(* IEC 61131-3 sources: SmartHomeNew/, 564 files *)

(* ---- E_Heating_Policy_Mode.typ ---- *)
TYPE E_Heating_Policy_Mode :
(
    HPM_NORMAL,
    HPM_DEGRADED,
    HPM_FREEZE_PROTECT,
    HPM_MAINTENANCE,
    HPM_SAFETY_BLOCK,
    HPM_FAULT_ISOLATION
);
END_TYPE

(* ---- E_Modbus_SysCom_Backend_State.dut ---- *)
TYPE E_Modbus_SysCom_Backend_State :
(
    MB_SYSCOM_CLOSED := 0,
    MB_SYSCOM_OPENING := 1,
    MB_SYSCOM_ONLINE := 2,
    MB_SYSCOM_ERROR := 3,
    MB_SYSCOM_RECONNECT_WAIT := 4
);
END_TYPE

(* ---- E_Recovery_Phase.dut ---- *)
{attribute 'strict'}
TYPE E_Recovery_Phase :
(
    IDLE := 0,
    STABILIZING := 1,
    WAIT_MANUAL_CONFIRM := 2,
    RECOVERING := 3,
    COOLDOWN := 4,
    ABORTED := 5
) USINT;
END_TYPE

(* ---- E_Runtime_Observer_Deny_Reason.typ ---- *)
TYPE E_Runtime_Observer_Deny_Reason :
(
    RODR_NONE := 0,
    RODR_NO_ENABLE_REQUEST := 10,
    RODR_BOOTSTRAP_DISABLED := 100,
    RODR_PASSIVE_MODE_DISABLED := 110,
    RODR_READONLY_MODE_DISABLED := 120,
    RODR_GOVERNANCE_UNLOCKED := 130,
    RODR_RUNTIME_AUTHORITY_ENABLED := 140,
    RODR_WRITABLE_EXPORTS_ENABLED := 150
);
END_TYPE

(* ---- E_Safety_Mode.dut ---- *)
{attribute 'strict'}
TYPE E_Safety_Mode :
(
    NORMAL := 0,
    FIRE := 1,
    GAS := 2,
    WATER_LEAK := 3,
    GLOBAL_STOP := 4
) USINT;
END_TYPE

(* ---- E_SCENARIO_TYPE.dut ---- *)
{attribute 'strict'}
TYPE E_SCENARIO_TYPE :
(
    SCENARIO_NONE := 0,
    SCENARIO_MORNING := 1,
    SCENARIO_EVENING := 2,
    SCENARIO_AWAY := 3,
    SCENARIO_PARTY := 4,
    SCENARIO_SLEEP := 5,
    SCENARIO_EMERGENCY := 6,
    SCENARIO_PRESENCE := 7
) USINT;
END_TYPE

(* ---- E_System_Reason_Code.dut ---- *)
{attribute 'strict'}
TYPE E_System_Reason_Code :
(
    REASON_NONE := 0,
    REASON_USER := 1,
    REASON_SAFETY := 2,
    REASON_AUTOMATION := 3,
    REASON_INTERNAL := 4,
    REASON_SCENARIO_VENT_BOOST := 5
) USINT;
END_TYPE

(* ---- E_Trace_Layer.dut ---- *)
{attribute 'strict'}
TYPE E_Trace_Layer :
(
    TRACE_SYSTEM := 0,
    TRACE_SAFETY := 1,
    TRACE_HEATING := 2,
    TRACE_IO := 3,
    TRACE_SCENARIO := 4,
    TRACE_USER := 5
) USINT;
END_TYPE

(* ---- E_Trace_Source.dut ---- *)
{attribute 'strict'}
TYPE E_Trace_Source :
(
    SRC_MAIN := 0,
    SRC_IO := 1,
    SRC_DIAGNOSTICS := 2,
    SRC_HEATING := 3,
    SRC_SCENARIO := 4
) USINT;
END_TYPE

(* ---- E_Valve_Test_Result.dut ---- *)
{attribute 'strict'}
TYPE E_Valve_Test_Result :
(
    TEST_RESULT_NONE := 0,
    TEST_RESULT_PASSED := 1,
    TEST_RESULT_CURRENT_DEVIATION := 2,
    TEST_RESULT_TIME_DEVIATION := 3,
    TEST_RESULT_STALL := 4,
    TEST_RESULT_LIMIT_SWITCH_FAIL := 5,
    TEST_RESULT_ABORTED := 6
) USINT;
END_TYPE

(* ---- GVL_EXPLAINABILITY.gvl ---- *)
TYPE E_System_Reason_Code :
(
    REASON_NONE,
    REASON_FIRE,
    REASON_GAS,
    REASON_WATER_LEAK,
    REASON_GLOBAL_STOP,
    REASON_EVACUATION,
    REASON_RECOVERY_ACTIVE,
    REASON_SAFETY,
    REASON_USER_REQUEST,
    REASON_COMMAND_CLAMP,
    REASON_DOMAIN_PROJECTION,
    REASON_SCENARIO_NIGHT,
    REASON_SCENARIO_COMFORT,
    REASON_SCENARIO_ENERGY_SAVE,
    REASON_SCENARIO_AWAY,
    REASON_SCENARIO_PREHEAT,
    REASON_SCENARIO_ACCESS_SECURE,
    REASON_SCENARIO_VENT_BOOST
);
END_TYPE

VAR_GLOBAL
    G_Last_Global_Reason_Code : E_System_Reason_Code := REASON_NONE;
    G_Last_Global_Reason_Text : STRING(255) := 'No active reason';
    G_Last_Safety_Mode : E_Safety_Mode := NORMAL;
    G_Last_Recovery_Phase : E_Recovery_Phase := IDLE;
    G_Last_Command_Source : STRING(80) := '';
    G_Last_Domain_Affected : STRING(80) := '';
    G_Last_Output_Affected : STRING(80) := '';
    G_Last_Update_MS : UDINT := 0;

    G_Behavior_Why_Active : STRING(255) := '';
    G_Heating_Why_Blocked : STRING(255) := '';
    G_Vent_Why_Stopped : STRING(255) := '';
    G_Water_Why_Closed : STRING(255) := '';
    G_Access_Why_Opened : STRING(255) := '';

    // Decision chain for HMI / engineering debug.
    G_Reason_Chain_Safety : STRING(80) := 'NORMAL';
    G_Reason_Chain_Behavior : STRING(120) := 'No behavior scenario active';
    G_Reason_Chain_Command : STRING(120) := 'Command OK';
    G_Reason_Chain_Output : STRING(120) := 'Outputs projected';
    G_Reason_Chain_Full : STRING(255) := 'NORMAL -> No behavior scenario active -> Command OK -> Outputs projected';
END_VAR

(* ---- GVL_SAFETY_RECOVERY.gvl ---- *)
TYPE E_Recovery_Phase :
(
    IDLE,
    STABILIZING,
    WAIT_MANUAL_CONFIRM,
    RECOVERING,
    COOLDOWN,
    ABORTED
);
END_TYPE

VAR_GLOBAL
    G_Recovery_Phase : E_Recovery_Phase := IDLE;
    G_Recovery_Active : BOOL := FALSE;
    G_Recovery_Requested : BOOL := FALSE;
    G_Recovery_Manual_Confirm : BOOL := FALSE;
    G_Recovery_Start_MS : UDINT := 0;
    G_Recovery_Stable_Since_MS : UDINT := 0;
    G_Recovery_Cooldown_Start_MS : UDINT := 0;
    G_Recovery_Exit_Allowed : BOOL := FALSE;
    G_Recovery_Abort_Reason : INT := 0; // 0=none, 1=safety active, 2=confidence low, 3=timeout
END_VAR

(* ---- GVL_SEMANTIC_EXECUTION_CONTROL.gvl ---- *)
TYPE E_SEMANTIC_EXECUTION_PATH : (
    FAST_PATH,
    NORMAL_PATH,
    DEFERRED_PATH,
    BACKGROUND_PATH
);
END_TYPE

VAR_GLOBAL
    // Semantic execution governance.
    Semantic_Execution_Control_Active : BOOL := TRUE;
    Semantic_Execution_Control_ReadOnly : BOOL := TRUE;

    // Canonical verification domains.
    Temporal_Verification_Domain_Active : BOOL := TRUE;
    Authority_Verification_Domain_Active : BOOL := TRUE;
    Physical_Verification_Domain_Active : BOOL := TRUE;
    Runtime_Verification_Domain_Active : BOOL := TRUE;
    Survivability_Verification_Domain_Active : BOOL := TRUE;

    // Deterministic semantic scheduling.
    Safety_Execution_Path : E_SEMANTIC_EXECUTION_PATH := FAST_PATH;
    Physical_Verification_Path : E_SEMANTIC_EXECUTION_PATH := FAST_PATH;
    Runtime_Verification_Path : E_SEMANTIC_EXECUTION_PATH := NORMAL_PATH;
    Diagnostics_Execution_Path : E_SEMANTIC_EXECUTION_PATH := DEFERRED_PATH;
    Trend_Analytics_Execution_Path : E_SEMANTIC_EXECUTION_PATH := BACKGROUND_PATH;

    // Semantic execution collapse prevention.
    Semantic_Execution_Fragmentation_Risk : BOOL := FALSE;
    Semantic_Cascade_Amplification_Risk : BOOL := FALSE;
    Semantic_Complexity_Ceiling_Reached : BOOL := FALSE;

    // Runtime semantic limits.
    Semantic_Chain_Depth_Limit_Reached : BOOL := FALSE;
    Verification_Fanout_Limit_Reached : BOOL := FALSE;
    Observability_Fanout_Limit_Reached : BOOL := FALSE;
    Lifecycle_Transition_Limit_Reached : BOOL := FALSE;

    // Runtime-governed complexity ceiling.
    Autonomous_Complexity_Ceiling_Enforced : BOOL := FALSE;
    Semantic_Scheduler_Active : BOOL := TRUE;

    Semantic_Execution_Control_Epoch : UDINT := 0;
END_VAR

(* ---- GVL_TRACE.gvl ---- *)
TYPE E_Trace_Layer :
(
    TRACE_SENSOR,
    TRACE_SCENARIO,
    TRACE_INTENT,
    TRACE_COMMAND,
    TRACE_DOMAIN,
    TRACE_IO,
    TRACE_SAFETY,
    TRACE_RECOVERY
);
END_TYPE

TYPE E_Trace_Source :
(
    SRC_NONE,
    SRC_SENSOR,
    SRC_USER,
    SRC_SCENARIO,
    SRC_SAFETY,
    SRC_RECOVERY,
    SRC_COMMAND,
    SRC_DOMAIN,
    SRC_IO
);
END_TYPE

TYPE ST_Trace_Entry :
STRUCT
    Timestamp_MS : UDINT;
    Layer : E_Trace_Layer;
    Source : E_Trace_Source;
    Reason_Code : E_System_Reason_Code;
    Value_Bool : BOOL;
    Value_Real : REAL;
    Text : STRING(120);
END_STRUCT
END_TYPE

VAR_GLOBAL
    G_Trace_Buffer : ARRAY[1..200] OF ST_Trace_Entry;
    G_Trace_Write_Index : INT := 1;
    G_Trace_Enabled : BOOL := TRUE;
END_VAR

(* ---- ST_Astro_Time.dut ---- *)
{attribute 'pack_mode' := '1'}
TYPE ST_Astro_Time :
STRUCT
    sunrise_ms : UDINT := 0;
    sunset_ms : UDINT := 0;
    is_daylight : BOOL := FALSE;
END_STRUCT
END_TYPE

(* ---- ST_BlackBox_Record.dut ---- *)
{attribute 'pack_mode' := '1'}
TYPE ST_BlackBox_Record :
STRUCT
    Timestamp : UDINT;
    Gas_Methane_LEL : REAL;
    Gas_CO_PPM : REAL;
    Flood_Active : BOOL;
    Fire_Active : BOOL;
    Valve_Gas_Status : BYTE;
    Valve_Water_Status : BYTE;
    PLC_Active_ID : BYTE;
    System_Mode : BYTE; // Encoded E_System_Operating_Mode for diagnostics
    First_Fault_Type : BYTE; // 1=IO,2=Sensor,3=Comm,4=Subsystem
    First_Fault_Source : BYTE; // 1=Heating,2=DHW,3=Ventilation,4=Lighting,5=Access
    First_Fault_Active : BOOL;
    System_Severity : BYTE;
    Root_Cause      : BYTE;
    Watchdog_Fault  : BOOL; // Latched root cause active

END_STRUCT
END_TYPE

(* ---- ST_Boiler_Status.dut ---- *)
{attribute 'pack_mode' := '1'}
TYPE ST_Boiler_Status :
STRUCT
    Active : BOOL;
    Running : BOOL;
    Warning : BOOL;
    Error : BOOL;
    Error_ID : WORD;

    // Boiler thermal/runtime information
    Power_Percent : REAL;
    Current_Power : REAL;
    Work_Seconds : UDINT;
    Work_Hours : REAL;
    Resource_Percent : REAL := 100.0;
    Last_Start : DT;

    // OpenTherm transport observability
    OT_Online : BOOL;
    OT_Command_Valid : BOOL;
    OT_Transport_Degraded : BOOL;
    OT_Adapter_Error : BOOL;

    // Semantic cascade/explainability state
    Available : BOOL;
    Selected_By_Cascade : BOOL;
    Flame_Missing : BOOL;
    Transport_Missing : BOOL;
    Ignition_Timeout : BOOL;
    Degraded : BOOL;
END_STRUCT
END_TYPE

(* ---- ST_Config_Activation_State.dut ---- *)
TYPE ST_Config_Activation_State :
STRUCT
    Runtime_Valid : BOOL;
    Runtime_System_Time_MS : UDINT;

    Active_Version : UDINT;
    Staged_Version : UDINT;
    Previous_Stable_Version : UDINT;

    Staged_Config_Valid : BOOL;
    Activation_Requested : BOOL;
    Activation_Allowed : BOOL;
    Activation_Blocked : BOOL;
    Rollback_Requested : BOOL;
    Rollback_Available : BOOL;
    Rollback_Active : BOOL;

    Config_Quarantine_Active : BOOL;
    Migration_Required : BOOL;
    Migration_Compatible : BOOL;

    Status_Code : UINT;
    Status_Text : STRING(160);
END_STRUCT
END_TYPE

(* ---- ST_Debug_Log_Record.dut ---- *)
{attribute 'pack_mode' := '1'}
TYPE ST_Debug_Log_Record :
STRUCT
    timestamp_ms : UDINT;
    level : BYTE; // E_Debug_Log_Level
    source_id : BYTE;
    event_code : WORD;
    value_int : UDINT;
    value_real : REAL;
    text : STRING(80);
    crc32 : DWORD;
END_STRUCT
END_TYPE

(* ---- ST_Distributed_Projection_Ownership.dut ---- *)
TYPE ST_Distributed_Projection_Ownership :
STRUCT
    Ownership_Valid : BOOL;
    Runtime_System_Time_MS : UDINT;

    Projection_Id : UINT;
    Projection_Class : UINT;

    Owner_Controller_Id : UINT;
    Owner_Runtime_Node_Id : UINT;
    Owner_Authority_Domain_Id : UINT;

    Ownership_Granted : BOOL;
    Ownership_Revoked : BOOL;
    Ownership_Conflict : BOOL;
    Ownership_Stale : BOOL;

    Projection_Active : BOOL;
    Projection_Blocked : BOOL;

    Distributed_Execution_Allowed : BOOL;
    Distributed_Recovery_Allowed : BOOL;

    Status_Code : UINT;
    Status_Text : STRING(160);
END_STRUCT
END_TYPE

(* ---- ST_Distributed_Runtime_Node_State.dut ---- *)
TYPE ST_Distributed_Runtime_Node_State :
STRUCT
    Runtime_Valid : BOOL;
    Runtime_System_Time_MS : UDINT;

    Controller_Id : UINT;
    Runtime_Node_Id : UINT;
    Authority_Domain_Id : UINT;
    Topology_Domain_Id : UINT;

    Node_Online : BOOL;
    Node_Degraded : BOOL;
    Node_Quarantined : BOOL;
    Node_Backup_Mode : BOOL;
    Node_Observer_Mode : BOOL;

    Authority_Allowed : BOOL;
    Authority_Revoked : BOOL;
    Authority_Master : BOOL;
    Authority_Backup : BOOL;

    Replication_Healthy : BOOL;
    Replication_Timeout : BOOL;
    Split_Brain_Suspected : BOOL;

    Restart_Continuity_Valid : BOOL;
    Quarantine_State_Replicated : BOOL;
    Recovery_State_Replicated : BOOL;

    Status_Code : UINT;
    Status_Text : STRING(160);
END_STRUCT
END_TYPE

(* ---- ST_Distributed_Topology_Domain.dut ---- *)
TYPE ST_Distributed_Topology_Domain :
STRUCT
    Domain_Valid : BOOL;
    Domain_Id : UINT;
    Controller_Id : UINT;
    Runtime_Node_Id : UINT;

    Authority_Owner : BOOL;
    Backup_Owner : BOOL;
    Observer_Only : BOOL;

    Domain_Online : BOOL;
    Domain_Degraded : BOOL;
    Domain_Quarantined : BOOL;

    Cross_Node_Dependencies : BOOL;
    Remote_Valve_Group_Required : BOOL;
    Remote_Recovery_Required : BOOL;

    Distributed_Path_Valid : BOOL;
    Distributed_Projection_Allowed : BOOL;

    Status_Code : UINT;
    Status_Text : STRING(160);
END_STRUCT
END_TYPE

(* ---- ST_EVENT.dut ---- *)
TYPE ST_EVENT :
STRUCT
    Event_ID    : UDINT;
    Event_Type  : UINT;
    Timestamp   : UDINT;
    Param1      : UDINT;
    Param2      : UDINT;
END_STRUCT
END_TYPE

(* ---- ST_Flood_Config.dut ---- *)
{attribute 'pack_mode' := '1'}
TYPE ST_Flood_Config :
STRUCT
    Emergency_Two_Stage_Enabled : BOOL := TRUE;
    Valve_Test_Period_Days : UINT := 7;
    Current_Threshold_MA : REAL := 500.0;
    sensor_to_valve_map : ARRAY[1..GVL_CONSTANTS.C_MAX_FLOOD_SENSORS] OF INT := [1, 1, 1, 1, 2, 2, 2, 2, 3, 3, 3, 3]; // 1: ХВС, 2: ГВС, 3: Оба
END_STRUCT
END_TYPE

(* ---- ST_Heating_Command.st ---- *)
TYPE ST_Heating_Command :
STRUCT
    Enable              : BOOL;
    Target_Temperature  : REAL;
    Priority            : INT; // higher = stronger
END_STRUCT
END_TYPE

(* ---- ST_Heating_Runtime_Adaptive_Intelligence.dut ---- *)
TYPE ST_Heating_Runtime_Adaptive_Intelligence :
STRUCT
    // ======================================================
    // Adaptive lifecycle
    // ======================================================
    Intelligence_Active : BOOL;
    Intelligence_Degraded : BOOL;
    Intelligence_Critical : BOOL;

    // ======================================================
    // Adaptive supervision confidence
    // ======================================================
    Supervision_Confidence : UINT;
    Confidence_Degraded : BOOL;

    // ======================================================
    // Adaptive runtime risk
    // ======================================================
    Adaptive_Runtime_Risk : UINT;
    Adaptive_Runtime_Stability : UINT;

    // ======================================================
    // Adaptive anomaly weighting
    // ======================================================
    Runtime_Anomaly_Weight : UINT;
    Cascade_Anomaly_Weight : UINT;
    OpenTherm_Anomaly_Weight : UINT;
    Diagnostics_Anomaly_Weight : UINT;

    // ======================================================
    // Predictive correlation weighting
    // ======================================================
    Predictive_Correlation_Score : UINT;
    Predictive_Correlation_Degraded : BOOL;

    // ======================================================
    // Adaptive integrity
    // ======================================================
    Sequencing_Confidence : UINT;
    Ownership_Confidence : UINT;
    Synchronization_Confidence : UINT;

    // ======================================================
    // Adaptive status
    // ======================================================
    Status_Code : UINT;
    Status_Text : STRING(128);
END_STRUCT
END_TYPE

(* ---- ST_Heating_Runtime_Blackbox_Timeline.dut ---- *)
TYPE ST_Heating_Runtime_Blackbox_Timeline :
STRUCT
    // ======================================================
    // Blackbox events
    // ======================================================
    Events : ARRAY[1..256] OF ST_Heating_Runtime_Blackbox_Event;

    // ======================================================
    // Timeline state
    // ======================================================
    Write_Index : UINT;
    Event_Count : UINT;
    Timeline_Overflow : BOOL;

    // ======================================================
    // Runtime forensic state
    // ======================================================
    Reconstruction_Active : BOOL;
    Replay_Active : BOOL;
    Root_Cause_Reconstructed : BOOL;

    // ======================================================
    // Timeline integrity
    // ======================================================
    Sequencing_Valid : BOOL;
    Ownership_Valid : BOOL;
    Synchronization_Valid : BOOL;

    // ======================================================
    // Timeline status
    // ======================================================
    Status_Code : UINT;
    Status_Text : STRING(128);
END_STRUCT
END_TYPE

(* ---- ST_Heating_Runtime_Causality_Edge.dut ---- *)
TYPE ST_Heating_Runtime_Causality_Edge :
STRUCT
    // ======================================================
    // Edge topology
    // ======================================================
    Source_Node_ID : UINT;
    Target_Node_ID : UINT;

    // ======================================================
    // Edge lifecycle
    // ======================================================
    Edge_Active : BOOL;
    Propagation_Detected : BOOL;

    // ======================================================
    // Propagation state
    // ======================================================
    Runtime_Propagation : BOOL;
    Cascade_Propagation : BOOL;
    OpenTherm_Propagation : BOOL;
    Diagnostics_Propagation : BOOL;

    // ======================================================
    // Propagation integrity
    // ======================================================
    Sequencing_Propagation : BOOL;
    Ownership_Propagation : BOOL;
    Synchronization_Propagation : BOOL;

    // ======================================================
    // Edge severity
    // ======================================================
    Severity_Level : UINT;
    Critical_Path : BOOL;

    // ======================================================
    // Edge status
    // ======================================================
    Status_Code : UINT;
    Status_Text : STRING(128);
END_STRUCT
END_TYPE

(* ---- ST_Heating_Runtime_Integration_Bridge.dut ---- *)
TYPE ST_Heating_Runtime_Integration_Bridge :
STRUCT
    // ======================================================
    // Runtime orchestration shell state
    // ======================================================
    Shell_Ready : BOOL;
    Shell_Fault : BOOL;
    Shell_Contract_Valid : BOOL;

    // ======================================================
    // Observation-only integration readiness
    // ======================================================
    Allow_DHW_Integration : BOOL;
    Allow_Heating_Integration : BOOL;
    Allow_Diagnostics_Integration : BOOL;
    Allow_Output_Projection_Integration : BOOL;

    // ======================================================
    // Runtime ownership integrity
    // ======================================================
    Runtime_Ownership_Valid : BOOL;
    Diagnostics_Ownership_Valid : BOOL;
    Explainability_Ownership_Valid : BOOL;
    OpenTherm_Ownership_Valid : BOOL;
    Cascade_Ownership_Valid : BOOL;
    Safety_Ownership_Valid : BOOL;

    // ======================================================
    // Runtime sequencing integrity
    // ======================================================
    DHW_Before_Heating_Valid : BOOL;
    Diagnostics_After_Publication_Valid : BOOL;
    Output_Projection_Last_Valid : BOOL;

    // ======================================================
    // Governance lock state
    // Observation only.
    // No migration authority exists in supervision.
    // ======================================================
    Governance_Locked : BOOL;
    Runtime_Attachment_Allowed : BOOL;
    Runtime_Attachment_Active : BOOL;

    // ======================================================
    // Runtime integration status
    // ======================================================
    Integration_Status_Code : UINT;
    Integration_Status_Text : STRING(128);

    // ======================================================
    // Runtime integration visibility
    // ======================================================
    Diagnostics_Visible : BOOL;
    Explainability_Visible : BOOL;

    // ======================================================
    // Runtime phase synchronization
    // ======================================================
    Current_Phase : E_Heating_Runtime_Phase;
    Runtime_Synchronized : BOOL;
END_STRUCT
END_TYPE

(* ---- ST_Heating_Runtime_Meta_Supervision.dut ---- *)
TYPE ST_Heating_Runtime_Meta_Supervision :
STRUCT
    // ======================================================
    // Meta-supervision lifecycle
    // ======================================================
    Meta_Supervision_Active : BOOL;
    Meta_Supervision_Degraded : BOOL;
    Meta_Supervision_Critical : BOOL;

    // ======================================================
    // Supervision integrity
    // ======================================================
    Supervision_Integrity_Valid : BOOL;
    Supervision_Integrity_Score : UINT;

    // ======================================================
    // Adaptive supervision drift
    // ======================================================
    Adaptive_Drift_Detected : BOOL;
    Adaptive_Drift_Score : UINT;

    // ======================================================
    // Predictive confidence decay
    // ======================================================
    Confidence_Decay_Detected : BOOL;
    Confidence_Decay_Score : UINT;

    // ======================================================
    // Intelligence consistency
    // ======================================================
    Intelligence_Consistency_Valid : BOOL;
    Intelligence_Consistency_Score : UINT;

    // ======================================================
    // Meta integrity
    // ======================================================
    Sequencing_Meta_Valid : BOOL;
    Ownership_Meta_Valid : BOOL;
    Synchronization_Meta_Valid : BOOL;

    // ======================================================
    // Meta-supervision status
    // ======================================================
    Status_Code : UINT;
    Status_Text : STRING(128);
END_STRUCT
END_TYPE

(* ---- ST_Heating_Runtime_Predictive_State.dut ---- *)
TYPE ST_Heating_Runtime_Predictive_State :
STRUCT
    // ======================================================
    // Predictive analytics visibility
    // Passive analytics only.
    // No predictive authority exists.
    // ======================================================
    Predictive_Analytics_Visible : BOOL;
    Predictive_Analytics_Degraded : BOOL;
    Predictive_Analytics_Attention : BOOL;

    // ======================================================
    // Runtime stability observation
    // ======================================================
    Runtime_Stable : BOOL;
    Runtime_Stability_Score : UINT;

    // ======================================================
    // Runtime degradation observation
    // ======================================================
    Runtime_Degradation_Observation : UINT;
    Runtime_Failure_Observation : UINT;

    // ======================================================
    // Source stability observation
    // Passive aggregate only.
    // Per-circuit details remain in GVL_Heating_Source_Stability.G_State.
    // ======================================================
    Source_Instability_Observation : UINT;
    Source_Instability_Attention : BOOL;
    Source_Oscillation_Trend_Visible : BOOL;
    Source_Degraded_Trend_Visible : BOOL;
    Source_Loss_Trend_Visible : BOOL;

    // ======================================================
    // Cascade observational analytics
    // ======================================================
    Cascade_Degradation_Observation : UINT;
    Cascade_Degraded_Trend_Visible : BOOL;

    // ======================================================
    // OpenTherm observational analytics
    // ======================================================
    OpenTherm_Instability_Observation : UINT;
    OpenTherm_Degraded_Trend_Visible : BOOL;

    // ======================================================
    // Runtime integrity observation
    // ======================================================
    Sequencing_Observation : UINT;
    Ownership_Observation : UINT;
    Synchronization_Observation : UINT;

    // ======================================================
    // Predictive analytics status
    // ======================================================
    Status_Code : UINT;
    Status_Text : STRING(128);
END_STRUCT
END_TYPE

(* ---- ST_Heating_Runtime_Source_Instability_State.dut ---- *)
TYPE ST_Heating_Runtime_Source_Instability_State :
STRUCT
    // Canonical predictive observability contract.
    // Observation-only.

    Visible : BOOL;

    // Edge counters
    Source_Switch_Count : UINT;
    Fallback_Activation_Count : UINT;
    Fallback_Recovery_Count : UINT;
    Source_Loss_Count : UINT;

    // Trend semantics
    Degraded_Trend_Visible : BOOL;
    Recovery_Trend_Visible : BOOL;
    Oscillation_Detected : BOOL;
    Instability_Attention : BOOL;

    // Predictive semantics
    Instability_Score : REAL;
    Confidence_Volatility : REAL;
    Source_Trust_Trend : REAL;

    // Explainability
    Status_Code : UINT;
    Status_Text : STRING(128);
    Last_Observation_MS : UDINT;
END_STRUCT
END_TYPE

(* ---- ST_Heating_Runtime_Supervisory_Publication.dut ---- *)
TYPE ST_Heating_Runtime_Supervisory_Publication :
STRUCT
    // Canonical supervisory publication surface.
    // Passive publication only.
    // No runtime authority.

    Supervisory_Visible : BOOL;

    // Predictive aggregation
    Predictive_State : ST_Heating_Runtime_Predictive_State;

    // Runtime observation
    Runtime_Degraded : BOOL;
    Runtime_Fault : BOOL;

    // Source instability aggregation
    Source_Instability_Attention : BOOL;
    Source_Oscillation_Trend_Visible : BOOL;

    // Explainability aggregation
    Explainability_Degraded : BOOL;
    Diagnostics_Degraded : BOOL;

    // Causality aggregation
    Causality_Active : BOOL;
    Propagation_Detected : BOOL;

    // Reconstruction aggregation
    Reconstruction_Visible : BOOL;

    // Supervisory publication status
    Status_Code : UINT;
    Status_Text : STRING(128);
END_STRUCT
END_TYPE

(* ---- ST_Heating_Schedule_Event.dut ---- *)
{attribute 'pack_mode' := '1'}
TYPE ST_Heating_Schedule_Event :
STRUCT
    Enabled : BOOL := FALSE;
    Comfort_Time_MS : UDINT := 28800000; // 08:00 from midnight
    Weekday_Mask : BYTE := 127; // bit0=Mon ... bit6=Sun
    Preheat_Boost : REAL := 0.5;
END_STRUCT
END_TYPE

(* ---- ST_HMI_Config_Workflow_State.dut ---- *)
TYPE ST_HMI_Config_Workflow_State :
STRUCT
    Runtime_Valid : BOOL;
    Runtime_System_Time_MS : UDINT;

    Editor_Open : BOOL;
    Edit_Session_Active : BOOL;
    Draft_Dirty : BOOL;

    Validation_Requested : BOOL;
    Validation_OK : BOOL;
    Validation_Failed : BOOL;
    Validated_Draft_Version : UDINT;
    Validation_Last_Run_MS : UDINT;
    Validation_Result_Seq : UDINT;

    Activation_Requested : BOOL;
    Activation_Allowed : BOOL;
    Activation_Blocked : BOOL;

    Rollback_Requested : BOOL;
    Rollback_Allowed : BOOL;

    Reset_Default_Requested : BOOL;
    Reset_Default_Allowed : BOOL;

    Operator_Ack_Required : BOOL;
    Service_Mode_Required : BOOL;
    Quarantine_Visible : BOOL;

    Active_Version : UDINT;
    Draft_Version : UDINT;
    Last_Stable_Version : UDINT;
    Topology_Draft_Version : UDINT;
    Validated_Topology_Version : UDINT;
    Topology_Activation_Required : BOOL;
    Topology_Validation_OK : BOOL;

    Status_Code : UINT;
    Status_Text : STRING(160);
END_STRUCT
END_TYPE

(* ---- ST_OpenTherm_Status.dut ---- *)
TYPE ST_OpenTherm_Status :
STRUCT
    Raw_Heartbeat : UDINT;
    Raw_Ack_Seq : UDINT;
    Raw_Online : BOOL;
    Raw_Error : BOOL;
    Raw_Flame : BOOL;
    Raw_Modulation_x10 : UINT;
    Raw_Boiler_Temp_x10 : INT;
    Raw_Status_Word : WORD;
    Raw_Error_Code : WORD;

    Adapter_Online : BOOL;
    Adapter_Error : BOOL;
    Command_Ack : BOOL;
    Command_Timeout : BOOL;
    Heartbeat_Timeout : BOOL;

    Last_Heartbeat : UDINT;
    Last_Heartbeat_MS : UDINT;

    Adapter_State : E_OpenTherm_Adapter_State;
    Error_State : E_OpenTherm_Error;
END_STRUCT
END_TYPE

(* ---- ST_Predictive_Diagnostics_State.dut ---- *)
TYPE ST_Predictive_Diagnostics_State :
STRUCT
    Runtime_Valid : BOOL;
    Runtime_System_Time_MS : UDINT;

    Device_Id : UINT;
    Device_Class : UINT;
    Valve_Group_Id : UINT;

    Failure_Count : UINT;
    Timeout_Count : UINT;
    Conflict_Count : UINT;
    Recovery_Denied_Count : UINT;

    Wear_Score : REAL;
    Reliability_Score : REAL;
    Intermittent_Fault_Suspected : BOOL;
    Degradation_Accumulating : BOOL;

    Service_Recommended : BOOL;
    Service_Urgent : BOOL;
    Predictive_Quarantine_Recommended : BOOL;

    Status_Code : UINT;
    Status_Text : STRING(160);
END_STRUCT
END_TYPE

(* ---- ST_Runtime_Node_Session.dut ---- *)
TYPE ST_Runtime_Node_Session :
STRUCT
    Session_Valid : BOOL;
    Session_Id : UDINT;
    Session_Start_MS : UDINT;
    Last_Heartbeat_MS : UDINT;

    Controller_Id : UINT;
    Runtime_Node_Id : UINT;

    Session_Connected : BOOL;
    Session_Stale : BOOL;
    Session_Reconnect_Required : BOOL;
    Session_Quarantined : BOOL;

    Transport_Healthy : BOOL;
    Runtime_Replication_Healthy : BOOL;

    Authority_Granted : BOOL;
    Authority_Revoked : BOOL;

    Status_Code : UINT;
    Status_Text : STRING(160);
END_STRUCT
END_TYPE

(* ---- ST_Runtime_Restart_Continuity_State.dut ---- *)
TYPE ST_Runtime_Restart_Continuity_State :
STRUCT
    Runtime_Valid : BOOL;
    Runtime_System_Time_MS : UDINT;

    Cold_Start_Detected : BOOL;
    Warm_Restart_Detected : BOOL;
    Restore_Requested : BOOL;
    Restore_Allowed : BOOL;
    Restore_Blocked : BOOL;
    Restore_Completed : BOOL;

    Retained_State_Valid : BOOL;
    Topology_Restore_Valid : BOOL;
    Config_Restore_Valid : BOOL;
    Recovery_Restore_Valid : BOOL;
    Quarantine_Restore_Valid : BOOL;

    Active_Config_Version : UDINT;
    Restored_Config_Version : UDINT;
    Last_Stable_Config_Version : UDINT;

    Post_Restart_Validation_Required : BOOL;
    Post_Restart_Validation_OK : BOOL;
    Post_Restart_Validation_Failed : BOOL;

    Safe_Mode_Required : BOOL;
    Operator_Ack_Required : BOOL;

    Status_Code : UINT;
    Status_Text : STRING(160);
END_STRUCT
END_TYPE

(* ---- ST_Scenario_Stats.dut ---- *)
TYPE ST_Scenario_Stats :
STRUCT
    Activations : UDINT;
    Last_Activation : UDINT;
END_STRUCT
END_TYPE

(* ---- ST_Scenario_Transition_Config.dut ---- *)
{attribute 'pack_mode' := '1'}
TYPE ST_Scenario_Transition_Config :
STRUCT
    current_scenario : E_SCENARIO_TYPE;
    target_scenario : E_SCENARIO_TYPE;
    min_duration_minutes : UDINT := 5;
    transition_allowed : BOOL := FALSE;
END_STRUCT
END_TYPE

(* ---- ST_Security_Global_Config.dut ---- *)
{attribute 'pack_mode' := '1'}
TYPE ST_Security_Global_Config :
STRUCT
    PIN_Code : STRING(4) := '1234';
    Phones : ARRAY[1..GVL_CONSTANTS.C_MAX_SECURITY_PHONES] OF STRING(15);

    // Время на ввод PIN после нарушения периметра.
    // entry_delay_seconds оставлен как совместимое имя, pin_entry_timeout_seconds — явная настройка HMI.
    entry_delay_seconds : UDINT := 45;
    pin_entry_timeout_seconds : UDINT := 45;

    // Время выхода после постановки на охрану.
    exit_delay_seconds : UDINT := 60;

    alarm_duration_seconds : UDINT := 180;
    two_person_timeout_seconds : UDINT := 120;
    max_access_attempts : BYTE := 3;

    // Комбинированная тревога: 2 и более независимых датчика за окно времени — тревога без задержки.
    combined_alarm_window_seconds : UDINT := 10;

    // Краткосрочная охрана с открытыми окнами.
    // Двери всё равно блокируют постановку. Разрешённые открытые окна игнорируются
    // до первого закрытия и не дают тревогу при автоматическом повышении уровня отъезда.
    allow_short_away_open_windows : BOOL := FALSE;

    auto_arm_enabled : BOOL := FALSE;
    auto_arm_time_ms : UDINT := 0;
    enable_2fa : BOOL := TRUE; // Включение/отключение двухфакторной аутентификации
    gate_open_pulse_ms : UDINT := GVL_CONSTANTS.C_MS_IN_SECOND;
    wicket_open_pulse_ms : UDINT := GVL_CONSTANTS.C_MS_IN_SECOND;
    lock_open_pulse_ms : UDINT := GVL_CONSTANTS.C_MS_IN_SECOND;
    lock_close_pulse_ms : UDINT := GVL_CONSTANTS.C_MS_IN_SECOND;

    // Байпасы зон
    bypass_motion : ARRAY[1..16] OF BOOL;
    bypass_doors : ARRAY[1..GVL_CONSTANTS.C_MAX_DOOR_SENSORS] OF BOOL;
    bypass_windows : ARRAY[1..16] OF BOOL;
END_STRUCT
END_TYPE

(* ---- ST_Socket_Command_V2.dut ---- *)
TYPE ST_Socket_Command_V2 : STRUCT
    Target_State : BOOL;
END_STRUCT
END_TYPE

(* ---- ST_Socket_State_V2.dut ---- *)
TYPE ST_Socket_State_V2 : STRUCT
    Is_On : BOOL;
    Safety_Blocked : BOOL;
END_STRUCT
END_TYPE

(* ---- ST_State_Snapshot.dut ---- *)
{attribute 'pack_mode' := '1'}
TYPE ST_State_Snapshot :
STRUCT
    timestamp_ms : UDINT := 0;
    operator_id : STRING(10) := '';
    scenario_id : E_SCENARIO_TYPE := E_SCENARIO_TYPE.SCENARIO_NONE;
    lighting_levels : ARRAY[1..GVL_CONSTANTS.C_MAX_LIGHTING_ZONES] OF BYTE;
    floor_heating_setpoints : ARRAY[1..GVL_CONSTANTS.C_MAX_HEATING_CIRCUITS] OF REAL;
    alarm_active : BOOL := FALSE;
    crc32 : DWORD := 0;
END_STRUCT
END_TYPE

(* ---- ST_System_Diagnostics.dut ---- *)
{attribute 'pack_mode' := '1'}
TYPE ST_System_Diagnostics :
STRUCT
    Freeze_Hardware_Event_Pending : BOOL;
    Freeze_Hardware_Event_Text : STRING(200);
    Backup_Pump_Fault : BOOL;
    Electric_Heater_Fault : BOOL;
    Backup_Pump_Recovered_After_Retry : BOOL;
    Electric_Heater_Recovered_After_Retry : BOOL;
    Backup_Pump_Out_Of_Service : BOOL;
    Electric_Heater_Out_Of_Service : BOOL;

    Pump_Exercise_Active : BOOL;
    Pump_Exercise_Failed : BOOL;
    Pump_Exercise_Last_Equipment : STRING(80);
    Pump_Exercise_Last_Result : STRING(120);
    Pump_Exercise_No_Feedback_Count : INT;
    Manifold_Pump_Exercise_Count : ARRAY[1..GVL_CONSTANTS.C_MAX_MANIFOLDS] OF UDINT;
    DHW_Heating_Pump_Exercise_Count : UDINT;
    DHW_Circ_Pump_Exercise_Count : UDINT;
    Backup_Pump_Exercise_Count : UDINT;
    Pump_Exercise_Event_Seq : UDINT;
    Pump_Exercise_Journal_1 : STRING(200);
    Pump_Exercise_Journal_2 : STRING(200);
    Pump_Exercise_Journal_3 : STRING(200);
    Pump_Exercise_Journal_Last_Seq : UDINT;

    Pump_Maintenance_Required : BOOL;
    Pump_Maintenance_Warning : BOOL;

    Manifold_Pump_Out_Of_Service : ARRAY[1..GVL_CONSTANTS.C_MAX_MANIFOLDS] OF BOOL;
    DHW_Heating_Pump_Out_Of_Service : BOOL;
    DHW_Circ_Pump_Out_Of_Service : BOOL;

    Maintenance_Last_Action : STRING(120);
    Operator_Action_Blocked : BOOL;
    Operator_Block_Reason : STRING(160);
    Operator_Last_Forbidden_Action : STRING(160);
    Operator_Journal_1 : STRING(200);
    Operator_Journal_2 : STRING(200);
    Operator_Journal_3 : STRING(200);
    Operator_Journal_Event_Seq : UDINT;
    Operator_Journal_Last_Seq : UDINT;

    Dangerous_Action_Pending_Confirm : BOOL;
    Dangerous_Action_Confirm_Text : STRING(160);
    Dangerous_Action_Confirm_Deadline_MS : UDINT;
    User_Access_Level_Active : INT;
    User_Access_Denied : BOOL;
    User_Access_Deny_Reason : STRING(160);

    Valve_Test_Mode_Active : BOOL;
    Valve_Test_Deadline_MS : UDINT;
    Valve_Test_Remaining_MS : UDINT;
    Valve_Test_Validation_OK : BOOL;
    Valve_Test_Validation_Text : STRING(160);
    Valve_Test_Forced_Close : BOOL;

    Water_Valve_Test_Mode_Active : BOOL;
    Water_Valve_Test_Deadline_MS : UDINT;
    Water_Valve_Test_Remaining_MS : UDINT;
    Water_Valve_Test_Validation_OK : BOOL;
    Water_Valve_Test_Validation_Text : STRING(160);
    Water_Valve_Test_Forced_Close : BOOL;
    Gas_Valve_Test_Mode_Active : BOOL;
    Gas_Valve_Test_Deadline_MS : UDINT;
    Gas_Valve_Test_Remaining_MS : UDINT;
    Gas_Valve_Test_Validation_OK : BOOL;
    Gas_Valve_Test_Validation_Text : STRING(160);
    Gas_Valve_Test_Forced_Close : BOOL;

    Active_Leak_Sensor_Index : INT;
    Active_Gas_Sensor_Index : INT;
    Active_Leak_Zone_Name : STRING(80);
    Active_Gas_Zone_Name : STRING(80);
    Water_Valve_Test_Context : STRING(160);
    Gas_Valve_Test_Context : STRING(160);

    Water_Recovery_Target_Zone_Index : INT;
    Gas_Recovery_Target_Zone_Index : INT;
    Water_Recovery_Selective_Allowed : BOOL;
    Gas_Recovery_Selective_Allowed : BOOL;
    Water_Recovery_Selective_Text : STRING(160);
    Gas_Recovery_Selective_Text : STRING(160);
    Water_Recovery_Physical_Active : BOOL;
    Water_Recovery_Physical_Zone_Name : STRING(80);

    Water_Zone_Open_Fault : ARRAY[1..32] OF BOOL;
    Water_Zone_Close_Fault : ARRAY[1..32] OF BOOL;
    Water_Zone_Open_Blocked : ARRAY[1..32] OF BOOL;
    Water_Open_Block_Active : BOOL;
    Water_Open_Block_Text : STRING(200);
    Water_Valve_Exercise_Last_Zone : INT;
    Water_Valve_Exercise_Last_Result : STRING(160);
    Water_Zone_Critical_Close_Fault : ARRAY[1..32] OF BOOL;
    Water_Close_Fault_Active : BOOL;
    Water_Close_Fault_Zone_Name : STRING(80);
    Water_Close_Fault_Text : STRING(200);
    Water_Zone_Close_Retry_Active : ARRAY[1..32] OF BOOL;
    Water_Zone_Close_Retry_Count : ARRAY[1..32] OF INT;
    Water_Zone_Close_Recovered_After_Retry : ARRAY[1..32] OF BOOL;
    Water_Localization_Failed : BOOL;
    Water_Main_Shutdown_Recommended : BOOL;
    Water_Escalation_Text : STRING(200);
    Alarm_Event_Pulse : BOOL;
    Alarm_Event_Code : UDINT;
    Alarm_Event_Value : REAL;
    Sensor_Fault : BOOL;
    IO_Offline : BOOL;
    Subsystem_Degraded : BOOL;

    Manifold_Pressure_Fault : ARRAY[1..GVL_CONSTANTS.C_MAX_MANIFOLDS] OF BOOL;
    Manifold_Pressure_Diag_Code : ARRAY[1..GVL_CONSTANTS.C_MAX_MANIFOLDS] OF WORD;
    Manifold_Pressure_Fault_Active : BOOL;
    Manifold_Pressure_First_Fault_Index : INT;
    Manifold_Pressure_Fault_Text : STRING(160);

    Manifold_Current_Fault : ARRAY[1..GVL_CONSTANTS.C_MAX_MANIFOLDS] OF BOOL;
    Manifold_Current_Diag_Code : ARRAY[1..GVL_CONSTANTS.C_MAX_MANIFOLDS] OF WORD;
    Manifold_Current_Fault_Active : BOOL;
    Manifold_Current_First_Fault_Index : INT;
    Manifold_Current_Fault_Text : STRING(160);

    Manifold_Return_Temp_Fault : ARRAY[1..GVL_CONSTANTS.C_MAX_MANIFOLDS] OF BOOL;
    Manifold_Return_Temp_Diag_Code : ARRAY[1..GVL_CONSTANTS.C_MAX_MANIFOLDS] OF WORD;
    Manifold_Return_Temp_Fault_Active : BOOL;
    Manifold_Return_Temp_First_Fault_Index : INT;
    Manifold_Return_Temp_Fault_Text : STRING(160);

    Manifold_Sensor_Fault_Count : ARRAY[1..GVL_CONSTANTS.C_MAX_MANIFOLDS] OF INT;
    Manifold_Sensor_Out_Of_Service : ARRAY[1..GVL_CONSTANTS.C_MAX_MANIFOLDS] OF BOOL;
    Manifold_Sensor_Out_Of_Service_Active : BOOL;
    Manifold_Sensor_First_OOS_Index : INT;
    Manifold_Sensor_OOS_Text : STRING(160);
END_STRUCT
END_TYPE

(* ---- ST_System_State_Snapshot.dut ---- *)
{attribute 'pack_mode' := '1'}
TYPE ST_System_State_Snapshot :
STRUCT
    // ======================================================
    // LEGACY DIRECT STATE REPLICATION SNAPSHOT
    // ======================================================
    // Used by legacy redundancy helpers that replicate/apply
    // domain state directly.
    //
    // This DUT is NOT the current distributed runtime protocol.
    // Current runtime-safe HA topology uses:
    // - GVL_PEER_SESSION
    // - GVL_HA_SESSION_REPLICATION
    // - PRG_Distributed_Peer_Ingestion
    // - PRG_Distributed_Commit_Ingestion
    //
    // Do not connect this snapshot path to MAIN as a parallel
    // HA runtime path without explicit barrier/governance review.
    // ======================================================

    System_Time_MS : UDINT;
    Current_Scenario : E_SCENARIO_TYPE;
    Security_Armed : BOOL;
    Active_Alarms : INT;
    // Критические состояния для синхронизации
    Zone_Valves : ARRAY[1..GVL_CONSTANTS.C_MAX_HEATING_CIRCUITS] OF BOOL;
    Manifold_Pumps : ARRAY[1..GVL_CONSTANTS.C_MAX_MANIFOLDS] OF BOOL;
    Lighting_States : ARRAY[1..32] OF BYTE;
    Blinds_Positions : ARRAY[1..GVL_CONSTANTS.C_MAX_BLINDS] OF BYTE;
    Socket_States : ARRAY[1..GVL_CONSTANTS.C_MAX_SOCKETS] OF BOOL;
    Gas_Valve_Closed : BOOL;
    Water_Valves_Closed : BOOL;
    Version : UDINT; // Версия состояния для разрешения конфликтов
END_STRUCT
END_TYPE

(* ---- ST_Trace_Entry.dut ---- *)
TYPE ST_Trace_Entry :
STRUCT
    Timestamp_MS : UDINT;
    Layer : E_Trace_Layer;
    Source : E_Trace_Source;
    Reason_Code : E_System_Reason_Code;
    Value_Bool : BOOL;
    Value_Real : REAL;
    Text : STRING(120);
END_STRUCT
END_TYPE

(* ---- ST_Trend_Data.dut ---- *)
{attribute 'pack_mode' := '1'}
TYPE ST_Trend_Data :
STRUCT
    config : ST_Trend_Config;
    record_count : UDINT;
    write_index : UDINT;
    sum_values : REAL;
    values : ARRAY[1..100] OF REAL;
    timestamps : ARRAY[1..100] OF UDINT;
    crc32 : DWORD;
END_STRUCT
END_TYPE

(* ---- ST_TwoFactor_Data.dut ---- *)
{attribute 'pack_mode' := '1'}
TYPE ST_TwoFactor_Data :
STRUCT
    operator_id : STRING(10);
    AuthMethod : BYTE; // E_TwoFactor_Method
    rfid_tag : STRING(20);
    totp_secret : STRING(32);
    last_modified : UDINT;
END_STRUCT
END_TYPE

(* ---- ST_Ventilation_Unit_Config.dut ---- *)
{attribute 'pack_mode' := '1'}
TYPE ST_Ventilation_Unit_Config :
STRUCT
    unit_id : BYTE := 0;
    unit_type : E_VENTILATION_UNIT_TYPE;
    location : E_VENTILATION_LOCATION;
    min_speed : BYTE := 20;
    max_speed : BYTE := 100;
    Threshold_Hum : REAL := 65.0;
    has_smoke_detector : BOOL := FALSE;
END_STRUCT
END_TYPE

(* ---- ST_Water_Actuator_Diagnostics_State.dut ---- *)
TYPE ST_Water_Actuator_Diagnostics_State :
STRUCT
    Runtime_Valid : BOOL;
    Runtime_System_Time_MS : UDINT;

    Valve_Group_Id : UINT;

    Travel_Active : BOOL;
    Travel_Timeout : BOOL;
    Stuck_Suspected : BOOL;
    Intermittent_Failure_Suspected : BOOL;

    Travel_Time_MS : UDINT;
    Failure_Count : UINT;

    Diagnostics_Degraded : BOOL;
    Escalation_Required : BOOL;

    Status_Code : UINT;
    Status_Text : STRING(128);
END_STRUCT
END_TYPE

(* ---- ST_Water_Hydraulic_Isolation_Group.dut ---- *)
TYPE ST_Water_Hydraulic_Isolation_Group :
STRUCT
    Runtime_Valid : BOOL;

    Isolation_Group_Id : UINT;
    Valve_Group_Id : UINT;
    Fallback_Domain_Id : UINT;

    Shared_Segment_Count : UINT;
    Shared_Sensor_Count : UINT;

    Isolation_Valid : BOOL;
    Isolation_Ambiguous : BOOL;

    Selective_Isolation_Allowed : BOOL;
    Global_Fallback_Required : BOOL;

    Status_Code : UINT;
    Status_Text : STRING(128);
END_STRUCT
END_TYPE

(* ---- ST_Water_Hydraulic_Topology_Node.dut ---- *)
TYPE ST_Water_Hydraulic_Topology_Node :
STRUCT
    Runtime_Valid : BOOL;

    Sensor_Id : UINT;
    Hydraulic_Zone_Id : UINT;
    Hydraulic_Segment_Id : UINT;
    Isolation_Group_Id : UINT;
    Valve_Group_Id : UINT;
    Fallback_Domain_Id : UINT;

    Mapping_Valid : BOOL;
    Mapping_Ambiguous : BOOL;
    Shared_Valve_Group : BOOL;

    Selective_Isolation_Allowed : BOOL;
    Global_Fallback_Required : BOOL;

    Status_Code : UINT;
    Status_Text : STRING(128);
END_STRUCT
END_TYPE

(* ---- ST_Water_Isolation_Runtime_State.dut ---- *)
TYPE ST_Water_Isolation_Runtime_State :
STRUCT
    // ==============================================================================
    // Water/Flood isolation semantic runtime state.
    // ==============================================================================
    //
    // Observe/publish-first governance contract.
    // Does NOT directly own valve outputs.
    // ==============================================================================

    Projection_Valid : BOOL;
    Projection_System_Time_MS : UDINT;

    // Isolation semantics.
    Isolation_Requested : BOOL;
    Selective_Isolation_Requested : BOOL;
    Global_Isolation_Requested : BOOL;

    // Topology semantics.
    Hydraulic_Zone_Id : UINT;
    Isolation_Group_Id : UINT;
    Valve_Group_Id : UINT;

    // Mapping validity.
    Mapping_Valid : BOOL;
    Fallback_To_Global_Required : BOOL;

    // Runtime compatibility visibility.
    Active_Global_Close_Path : BOOL;
    Active_Safety_Latch : BOOL;

    // Explainability.
    Reason_Code : UINT;
    Reason_Text : STRING(128);

    // Lifecycle edges.
    Isolation_Requested_Event : BOOL;
    Fallback_To_Global_Event : BOOL;

    // Governance identity.
    Supervisory_Observation_Only : BOOL;
END_STRUCT
END_TYPE

(* ---- ST_Water_Leak_Runtime_State.dut ---- *)
TYPE ST_Water_Leak_Runtime_State :
STRUCT
    // ==============================================================================
    // Canonical Water/Flood runtime semantic projection.
    //
    // Observe/publish-only contract.
    // Does NOT own valve authority or runtime arbitration.
    // ==============================================================================

    // Projection lifecycle.
    Projection_Valid : BOOL;
    Projection_System_Time_MS : UDINT;

    // Physical input source.
    Physical_Sensor_Index : UINT;
    Physical_Input_Valid : BOOL;

    // Logical leak semantics.
    Logical_Sensor_Valid : BOOL;
    Leak_Warning_Active : BOOL;
    Leak_Confirmed : BOOL;
    Leak_Cleared : BOOL;
    Leak_Degraded : BOOL;

    // Runtime-configurable topology semantics.
    Hydraulic_Zone_Id : UINT;
    Hydraulic_Segment_Id : UINT;
    Isolation_Group_Id : UINT;
    Valve_Group_Id : UINT;

    // Mapping semantics.
    Mapping_Valid : BOOL;
    Mapping_Missing : BOOL;
    Selective_Isolation_Possible : BOOL;
    Fallback_Global_Isolation_Required : BOOL;

    // Confidence / degradation.
    Leak_Confidence : REAL;
    Sensor_Quality_Valid : BOOL;
    Sensor_Stuck_Suspected : BOOL;
    Sensor_Noise_Suspected : BOOL;

    // Explainability.
    Reason_Code : UINT;
    Reason_Text : STRING(128);

    // Runtime lifecycle edges.
    Warning_Started_Event : BOOL;
    Leak_Confirmed_Event : BOOL;
    Leak_Cleared_Event : BOOL;
    Isolation_Requested_Event : BOOL;
    Mapping_Invalid_Event : BOOL;

    // Active runtime compatibility.
    Active_Safety_Leak_Latched : BOOL;
    Active_Global_Close_Path : BOOL;

    // Observability only.
    Supervisory_Observation_Only : BOOL;
END_STRUCT
END_TYPE

(* ---- ST_Water_Orchestration_Runtime_State.dut ---- *)
TYPE ST_Water_Orchestration_Runtime_State :
STRUCT
    Runtime_Valid : BOOL;
    Runtime_System_Time_MS : UDINT;

    Isolation_Sequence_Active : BOOL;
    Recovery_Sequence_Active : BOOL;

    Staged_Close_Required : BOOL;
    Staged_Open_Required : BOOL;

    Shared_Trunk_Sequencing : BOOL;

    Rollback_Required : BOOL;
    Escalation_Required : BOOL;

    Observation_Window_Active : BOOL;

    Sequencing_Valid : BOOL;

    Status_Code : UINT;
    Status_Text : STRING(128);
END_STRUCT
END_TYPE

(* ---- ST_Water_Output_Projection_State.dut ---- *)
TYPE ST_Water_Output_Projection_State :
STRUCT
    // Deterministic output projection contract.

    Projection_Valid : BOOL;
    Projection_System_Time_MS : UDINT;

    // Ownership.
    Output_Owner_Valid : BOOL;
    Output_Owner_Id : UINT;

    // Projection target.
    Valve_Id : UINT;
    Valve_Group_Id : UINT;

    // Authority source.
    Selective_Authority_Allowed : BOOL;
    Global_Fallback_Required : BOOL;
    Authority_Valid : BOOL;

    // Physical projection.
    Physical_Close_Project : BOOL;
    Physical_Open_Project : BOOL;

    // Reconciliation hooks.
    Expected_Closed : BOOL;
    Expected_Open : BOOL;
    Confirmed_Closed : BOOL;
    Confirmed_Open : BOOL;
    Feedback_Invalid : BOOL;

    // Arbitration validity.
    Projection_Allowed : BOOL;
    Projection_Denied : BOOL;

    // Explainability.
    Projection_Code : UINT;
    Projection_Text : STRING(128);

    // Lifecycle.
    Projection_Activated_Event : BOOL;
    Projection_Denied_Event : BOOL;
END_STRUCT
END_TYPE

(* ---- ST_Water_Output_Reconciliation_State.dut ---- *)
TYPE ST_Water_Output_Reconciliation_State :
STRUCT
    Runtime_Valid : BOOL;
    Runtime_System_Time_MS : UDINT;

    Valve_Group_Id : UINT;

    Projection_Active : BOOL;
    Runtime_Output_Active : BOOL;

    Expected_Closed : BOOL;
    Confirmed_Closed : BOOL;
    Feedback_Invalid : BOOL;

    Reconciliation_Healthy : BOOL;
    Projection_Runtime_Mismatch : BOOL;
    Projection_Confirmation_Mismatch : BOOL;

    Conflict_Detected : BOOL;
    Topology_Invalid : BOOL;

    Status_Code : UINT;
    Status_Text : STRING(128);
END_STRUCT
END_TYPE

(* ---- ST_Water_Recovery_Runtime_State.dut ---- *)
TYPE ST_Water_Recovery_Runtime_State :
STRUCT
    Runtime_Valid : BOOL;
    Runtime_System_Time_MS : UDINT;

    Recovery_Requested : BOOL;
    Recovery_Allowed : BOOL;
    Recovery_Denied : BOOL;

    Observation_Window_Active : BOOL;
    Unsafe_Recovery_Detected : BOOL;

    Valve_Degraded : BOOL;
    Confirmation_Healthy : BOOL;

    Recovery_Target_Valid : BOOL;

    Status_Code : UINT;
    Status_Text : STRING(128);
END_STRUCT
END_TYPE

(* ---- ST_Water_Topology_Validation_State.dut ---- *)
TYPE ST_Water_Topology_Validation_State :
STRUCT
    Runtime_Valid : BOOL;
    Runtime_System_Time_MS : UDINT;

    Sensor_Id : UINT;

    Topology_Valid : BOOL;
    Topology_Ambiguous : BOOL;
    Isolation_Path_Valid : BOOL;

    Shared_Valve_Group : BOOL;
    Missing_Valve_Group : BOOL;
    Invalid_Isolation_Group : BOOL;

    Selective_Isolation_Allowed : BOOL;
    Global_Fallback_Required : BOOL;

    Status_Code : UINT;
    Status_Text : STRING(128);
END_STRUCT
END_TYPE

(* ---- ST_Water_Valve_Feedback_State.dut ---- *)
TYPE ST_Water_Valve_Feedback_State :
STRUCT
    Runtime_Valid : BOOL;
    Runtime_System_Time_MS : UDINT;

    Valve_Group_Id : UINT;

    Feedback_Available : BOOL;

    Physical_Open_Feedback : BOOL;
    Physical_Closed_Feedback : BOOL;

    Confirmed_Open : BOOL;
    Confirmed_Closed : BOOL;

    Feedback_Invalid : BOOL;
    Feedback_Conflict : BOOL;
    Feedback_Timeout : BOOL;

    Travel_Timeout_Active : BOOL;
    Valve_Stuck_Suspected : BOOL;

    Valve_Degraded : BOOL;

    Status_Code : UINT;
    Status_Text : STRING(128);
END_STRUCT
END_TYPE

(* ---- ST_Water_Valve_Runtime_State.dut ---- *)
TYPE ST_Water_Valve_Runtime_State :
STRUCT
    // ==============================================================================
    // Water/Flood valve runtime semantic state.
    // ==============================================================================
    //
    // Observe-first valve governance contract.
    //
    // This contract does NOT directly own physical outputs.
    // ==============================================================================

    Runtime_Valid : BOOL;
    Runtime_System_Time_MS : UDINT;

    // Valve identity.
    Valve_Id : UINT;
    Valve_Group_Id : UINT;

    // Authority/runtime semantics.
    Close_Requested : BOOL;
    Open_Requested : BOOL;
    Global_Fallback_Request : BOOL;
    Selective_Authority_Allowed : BOOL;

    // Output/runtime visibility.
    Physical_Output_Active : BOOL;
    Output_Command_Projected : BOOL;

    // Confirmation semantics.
    Confirmation_Available : BOOL;
    Confirmed_Open : BOOL;
    Confirmed_Closed : BOOL;
    Confirmation_Timeout : BOOL;
    Feedback_Invalid : BOOL;

    // Diagnostics.
    Diagnostics_Available : BOOL;
    Valve_Healthy : BOOL;
    Valve_Stuck_Suspected : BOOL;
    Travel_Time_Degraded : BOOL;
    Current_Deviation_Detected : BOOL;

    // Governance/degraded semantics.
    Valve_Degraded : BOOL;
    Unsafe_Reopen_Denied : BOOL;
    Recovery_Allowed : BOOL;

    // Explainability.
    Status_Code : UINT;
    Status_Text : STRING(128);

    // Lifecycle edges.
    Close_Command_Event : BOOL;
    Open_Command_Event : BOOL;
    Confirmation_Lost_Event : BOOL;
    Valve_Degraded_Event : BOOL;
END_STRUCT
END_TYPE

(* ---- GVL_ACTUATOR_SEMANTIC_VERIFICATION.gvl ---- *)
VAR_GLOBAL
    // Global actuator semantic verification authority.
    Actuator_Semantic_Verification_Valid : BOOL := FALSE;
    Actuator_Semantic_Verification_Granted : BOOL := FALSE;
    Actuator_Semantic_Verification_Quarantine_Active : BOOL := TRUE;

    // Physical semantic realization proofs.
    Valve_Semantic_Realization_Valid : BOOL := FALSE;
    Relay_Semantic_Realization_Valid : BOOL := FALSE;
    Pump_Semantic_Realization_Valid : BOOL := FALSE;
    Fan_Semantic_Realization_Valid : BOOL := FALSE;
    Hydraulic_Response_Valid : BOOL := FALSE;

    // Closed-loop physical convergence.
    Physical_Effect_Converged : BOOL := FALSE;
    Actuation_Response_Temporal_Valid : BOOL := FALSE;
    Sensor_Confirmed_Execution_Valid : BOOL := FALSE;
    Semantic_Outcome_Aligned : BOOL := FALSE;

    // Semantic realization failure detectors.
    False_Positive_Actuation_Detected : BOOL := FALSE;
    Mechanical_NonRealization_Detected : BOOL := FALSE;
    Welded_Relay_Semantics_Detected : BOOL := FALSE;
    Hydraulic_NoEffect_Execution_Detected : BOOL := FALSE;
    Airflow_Realization_Mismatch_Detected : BOOL := FALSE;
    Physical_Convergence_Divergence_Detected : BOOL := FALSE;

    // Verification epochs.
    Actuator_Verification_Epoch : UDINT := 0;
    Actuator_Verification_Epoch_Coherent : BOOL := FALSE;

    // Temporal authority.
    Actuator_Verification_Last_Update_MS : UDINT := 0;
    Actuator_Verification_Lease_Expired : BOOL := TRUE;

    // Diagnostics.
    Actuator_Verification_Last_Error_Code : UDINT := 0;
    Actuator_Verification_Last_Error_Text : STRING(160) := '';
    Actuator_Verification_Invalidation_Count : UDINT := 0;
END_VAR

(* ---- GVL_ALARM.gvl ---- *)
{attribute 'qualified_only'}
VAR_GLOBAL
    G_Security_Armed : BOOL := FALSE; // Флаг: Система безопасности активирована
    G_Security_Siren : BOOL := FALSE;
    G_Global_Siren : BOOL := FALSE; // Глобальный флаг сирены от Alarm Manager
    G_Global_Critical : BOOL := FALSE;
    G_Global_Warning : BOOL := FALSE;
    G_Active_Alarm_Count : INT := 0;
    G_Unacked_Alarm_Count : INT := 0;
    G_Alarm_List : ARRAY[1..GVL_CONSTANTS.C_MAX_ALARMS] OF ST_Alarm_Record;
    G_Gas_Alarm_Active : BOOL := FALSE; // Флаг: Обнаружена критическая концентрация газа
    G_Gas_Fire_Siren : BOOL := FALSE;
    G_Fire_Alarm_Active : BOOL := FALSE; // Флаг: Сработали пожарные датчики
    G_Flood_Alarm_Active : BOOL := FALSE; // Флаг: Обнаружена протечка воды
    G_Security_Alarm : BOOL := FALSE; // Флаг: Тревога системы безопасности
END_VAR

VAR_GLOBAL RETAIN
    G_Next_Alarm_ID : UDINT := 1; // Глобальный счетчик ID тревог
END_VAR

(* ---- GVL_ALARM_AUDIBLE_ACK.gvl ---- *)
{attribute 'qualified_only'}
VAR_GLOBAL
    G_Ack_Request : BOOL := FALSE;
    G_Ack_Active : BOOL := FALSE;
    G_Ack_Start_MS : UDINT := 0;
    G_Ack_Expires_MS : UDINT := 0;
    G_Ack_Remaining_MS : UDINT := 0;
    G_Ack_Count_Current_Alarm : INT := 0;
    G_Ack_Limit_Reached : BOOL := FALSE;
    G_Last_Ack_Accepted : BOOL := FALSE;
    G_Last_Ack_Denied : BOOL := FALSE;
    G_Last_Denial_Code : UINT := 0;
    G_Last_Event_MS : UDINT := 0;
    G_Status_Text : STRING(200) := '';
END_VAR

(* ---- GVL_AUTHORITY_LINEAGE.gvl ---- *)
VAR_GLOBAL RETAIN
    // Persistent authority lineage.
    Authority_Lineage_Epoch : UDINT := 0;
    Authority_Lineage_Valid : BOOL := FALSE;

    // Persistence continuity proofs.
    Warm_Restart_Continuity_Valid : BOOL := FALSE;
    HA_Resume_Continuity_Valid : BOOL := FALSE;
    Retained_State_Integrity_Valid : BOOL := FALSE;

    // Replay/skew detection.
    Authority_Replay_Suspected : BOOL := FALSE;
    Retained_State_Skew_Detected : BOOL := FALSE;
    Partial_Authority_Resurrection_Detected : BOOL := FALSE;
    Epoch_Lineage_Discontinuity_Detected : BOOL := FALSE;

    // Last authoritative epochs.
    Last_Physical_Authority_Epoch : UDINT := 0;
    Last_Runtime_Epoch : UDINT := 0;
    Last_Output_Publication_Epoch : UDINT := 0;

    // Persistence metadata.
    Authority_Lineage_Boot_ID : UDINT := 0;
    Authority_Lineage_Last_Update_MS : UDINT := 0;

    // Diagnostics.
    Authority_Lineage_Last_Error_Code : UDINT := 0;
    Authority_Lineage_Last_Error_Text : STRING(160) := '';
    Authority_Lineage_Invalidation_Count : UDINT := 0;
END_VAR

(* ---- GVL_AUTHORITY_PROVENANCE_FABRIC.gvl ---- *)
VAR_GLOBAL
    // Global deterministic authority provenance governance.
    Authority_Provenance_Valid : BOOL := FALSE;
    Authority_Provenance_Granted : BOOL := FALSE;
    Authority_Provenance_Quarantine_Active : BOOL := TRUE;

    // Root authority authenticity proofs.
    Bootstrap_Authority_Authentic : BOOL := FALSE;
    Commissioning_Lineage_Traceable : BOOL := FALSE;
    Trust_Seed_Integrity_Valid : BOOL := FALSE;
    Root_Authority_Attribution_Coherent : BOOL := FALSE;
    Provenance_Causality_Grounded : BOOL := FALSE;

    // Long-term provenance integrity.
    Historical_Origin_Lineage_Valid : BOOL := FALSE;
    Distributed_Trust_Chain_Coherent : BOOL := FALSE;
    Authority_Origin_Continuity_Stable : BOOL := FALSE;
    Root_Identity_Cryptographic_Validity : BOOL := FALSE;

    // Authority-origin split-brain detectors.
    Bootstrap_Identity_Corruption_Detected : BOOL := FALSE;
    Forged_Authority_Root_Detected : BOOL := FALSE;
    Commissioning_Provenance_Gap_Detected : BOOL := FALSE;
    Trust_Seed_Impersonation_Detected : BOOL := FALSE;
    Origin_Authenticity_Erosion_Detected : BOOL := FALSE;
    Root_Lineage_Tampering_Detected : BOOL := FALSE;

    // Provenance epochs.
    Authority_Provenance_Epoch : UDINT := 0;
    Authority_Provenance_Epoch_Coherent : BOOL := FALSE;

    // Temporal authority.
    Authority_Provenance_Last_Update_MS : UDINT := 0;
    Authority_Provenance_Lease_Expired : BOOL := TRUE;

    // Diagnostics.
    Authority_Provenance_Last_Error_Code : UDINT := 0;
    Authority_Provenance_Last_Error_Text : STRING(160) := '';
    Authority_Provenance_Invalidation_Count : UDINT := 0;
END_VAR

(* ---- GVL_AWAY_RESTORE.gvl ---- *)
{attribute 'qualified_only'}
VAR_GLOBAL
    // Runtime-only snapshot for short-away restore.
    // Not RETAIN: this surface is intended for short departures within the
    // current runtime session. Safety layers still override restore outputs.
    G_Snapshot_Valid : BOOL := FALSE;
    G_Snapshot_Taken_MS : UDINT := 0;

    G_Lighting_Levels : ARRAY[1..GVL_CONSTANTS.C_MAX_LIGHT_ZONES] OF BYTE;
    G_Socket_States : ARRAY[1..GVL_CONSTANTS.C_MAX_SOCKETS] OF BOOL;

    G_Restore_Active : BOOL := FALSE;
    G_Restore_Progress : REAL := 0.0;
    G_Restore_Started_MS : UDINT := 0;
    G_Restore_Done : BOOL := FALSE;

    // One-cycle hold after progress reaches 1.0. Domain managers run later in
    // the cycle and must still see Active+Snapshot_Valid for final output apply.
    G_Restore_Finalize_Pending : BOOL := FALSE;
END_VAR

(* ---- GVL_BEHAVIOR_ADAPT.gvl ---- *)
VAR_GLOBAL
    // Scenario behavior weights.
    // Scalar fields are the active compile-safe source used by PRG_Scenario_Engine.
    G_Behavior_Weight_Comfort : REAL := 1.0;
    G_Behavior_Weight_Night : REAL := 1.0;
    G_Behavior_Weight_Preheat : REAL := 1.0;
    G_Behavior_Weight_VentBoost : REAL := 1.0;
    G_Behavior_Weight_AccessSecure : REAL := 1.0;

    G_Scenario_Stats : ARRAY[0..10] OF ST_Scenario_Stats;
    G_VentBoost_Zone_Adapt : ARRAY[1..GVL_CONSTANTS.C_MAX_ZONES] OF ST_Zone_Adapt_State;

    G_Adapt_Profile : E_Adapt_Profile := ADAPT_PROFILE_BALANCED;

    G_Adapt_Enabled : BOOL := TRUE;
    G_Adapt_Learning_Rate : REAL := 0.05;
    G_Adapt_Update_Threshold : INT := 5;

    G_Adapt_Min_Confidence : REAL := 0.30;
    G_Adapt_Default_Zone_Weight : REAL := 1.0;

    G_Confidence_Learning_Rate : REAL := 0.05;
    G_Decay_Factor : REAL := 0.995;

    G_Prev_Humidity : ARRAY[1..GVL_CONSTANTS.C_MAX_ZONES] OF REAL;
    G_Prev_Valid : ARRAY[1..GVL_CONSTANTS.C_MAX_ZONES] OF BOOL;
END_VAR
// >>> BULK_SYNC_ANCHOR: GVL_BEHAVIOR_ADAPT <<<

(* ---- GVL_CAUSAL_NARRATIVE_FABRIC.gvl ---- *)
VAR_GLOBAL
    Causal_Narrative_Active : BOOL := TRUE;
    Causal_Narrative_ReadOnly : BOOL := TRUE;

    Runtime_Narrative_Available : BOOL := FALSE;
    Recovery_Narrative_Available : BOOL := FALSE;
    Authority_Narrative_Available : BOOL := FALSE;
    Temporal_Narrative_Available : BOOL := FALSE;

    Narrative_Causality_Coherent : BOOL := FALSE;
    Narrative_Runtime_Alignment_Valid : BOOL := FALSE;

    Narrative_Opacity_Observed : BOOL := FALSE;
    Narrative_Gap_Observed : BOOL := FALSE;

    Runtime_Narrative_Code : STRING(255) := '';
    Recovery_Narrative_Code : STRING(255) := '';
    Authority_Narrative_Code : STRING(255) := '';

    Causal_Narrative_Epoch : UDINT := 0;
END_VAR

(* ---- GVL_Cluster_Runtime_FSM.gvl ---- *)
{attribute 'qualified_only'}
VAR_GLOBAL
    G_State_Startup : BOOL;
    G_State_Discovery : BOOL;
    G_State_Synchronization : BOOL;
    G_State_Operational : BOOL;
    G_State_Degraded : BOOL;
    G_State_Observer_Only : BOOL;
    G_State_Recovery_Lock : BOOL;
    G_State_Quarantine : BOOL;

    G_Runtime_Valid : BOOL;
    G_Last_Update_MS : UDINT;

    G_Status_Code : UINT;
    G_Status_Text : STRING(160);
END_VAR

(* ---- GVL_Cluster_Safety_Barrier.gvl ---- *)
{attribute 'qualified_only'}
VAR_GLOBAL
    G_Runtime_Valid : BOOL;
    G_Last_Update_MS : UDINT;

    G_Cluster_Execution_Blocked : BOOL;
    G_Authority_Downgraded : BOOL;
    G_Orchestration_Restricted : BOOL;

    G_Remote_Authority_Degraded : BOOL;
    G_Runtime_Bus_Degraded : BOOL;
    G_Projection_Ownership_Invalid : BOOL;
    G_Recovery_Lock_Active : BOOL;
    G_Deployment_Invalid : BOOL;

    G_Status_Code : UINT;
    G_Status_Text : STRING(160);
END_VAR

(* ---- GVL_CO_EXPOSURE.gvl ---- *)
{attribute 'qualified_only'}
VAR_GLOBAL
    G_CO_Max_PPM : REAL := 0.0;
    G_CO_Max_Sensor_Index : INT := 0;

    G_Level_30ppm_Active : BOOL := FALSE;
    G_Level_70ppm_Active : BOOL := FALSE;
    G_Level_400ppm_Active : BOOL := FALSE;

    G_Timer_30ppm_ET : TIME := T#0s;
    G_Timer_70ppm_ET : TIME := T#0s;
    G_Timer_400ppm_ET : TIME := T#0s;

    G_Timer_30ppm_Q : BOOL := FALSE;
    G_Timer_70ppm_Q : BOOL := FALSE;
    G_Timer_400ppm_Q : BOOL := FALSE;

    G_Warning_Active : BOOL := FALSE;
    G_Alarm_Active : BOOL := FALSE;
    G_Status_Text : STRING(160) := 'CO exposure idle';
    G_Last_Update_MS : UDINT := 0;
END_VAR

(* ---- GVL_COMMAND.gvl ---- *)
{attribute 'qualified_only'}
VAR_GLOBAL
    // ======================================================
    // LEGACY / OPERATOR COMMAND REQUEST SURFACE
    // ======================================================
    // This GVL is retained as a legacy/operator request surface.
    // Runtime operational command ownership lives in
    // GVL_COMMAND_SHADOW and is published by PRG_Command_Arbitration.
    //
    // Physical publication must not use GVL_COMMAND as final
    // output authority. Final actuator intent flows through:
    //   operator/safety/rules -> command arbitration -> GVL_COMMAND_SHADOW
    //   -> domain output GVLs -> PRG_IO_Write -> GVL_IO.
    //
    // Remaining direct GVL_COMMAND reads are limited to operator/service
    // functions such as reset, access level, confirmation and valve tests.
    // ======================================================

    G_Gas_Valve_Close : BOOL := FALSE;
    G_Boiler_Stop : BOOL := FALSE;
    G_Supply_100_Req : BOOL := FALSE;
    G_Supply_80_Req : BOOL := FALSE;
    G_Vent_PV3_Boost : BOOL := FALSE;
    G_Exhaust_100_Req : BOOL := FALSE;
    G_Vent_Stop : BOOL := FALSE;
    G_Close_Valve_35 : BOOL := FALSE;
    G_Close_Valve_36 : BOOL := FALSE;
    G_Gate_Open : BOOL;
    G_Wicket_Open : BOOL;
    G_Lock_1_Open : BOOL;
    G_Lock_1_Close : BOOL;
    G_Lock_2_Open : BOOL;
    G_Lock_2_Close : BOOL;
    G_Reset_Errors : BOOL := FALSE;
    G_Scenario_Request : E_SCENARIO_TYPE := E_SCENARIO_TYPE.SCENARIO_NONE;
    G_Scenario_Request_Operator : E_SCENARIO_TYPE := E_SCENARIO_TYPE.SCENARIO_NONE;

    G_Arm_Req : BOOL;
    G_Disarm_Req : BOOL;
    G_PIN_Code : STRING(4);
    G_RFID_Tag : STRING(20);
    G_2FA_Code_In : STRING(6);
    G_Send_2FA_Req : BOOL;
    G_2FA_Code_Out : STRING(6);
    G_Lighting_Override : ARRAY[1..GVL_CONSTANTS.C_MAX_LIGHT_ZONES] OF BYTE;
    G_Blinds_Override : ARRAY[1..GVL_CONSTANTS.C_MAX_BLINDS] OF BYTE;
    G_Socket_Override : ARRAY[1..GVL_CONSTANTS.C_MAX_SOCKETS] OF BOOL;
    CMD_Set_Manifold_Pump_In_Service : ARRAY[1..GVL_CONSTANTS.C_MAX_MANIFOLDS] OF BOOL;
    CMD_Set_DHW_Heating_Pump_In_Service : BOOL;
    CMD_Set_DHW_Circ_Pump_In_Service : BOOL;
    CMD_Dangerous_Action_Confirm : BOOL;
    CMD_Dangerous_Action_Request : BOOL;
    CMD_User_Access_Level : INT := 0;
    CMD_Valve_Test_Open : BOOL;
    CMD_Valve_Test_Close : BOOL;
    CMD_Valve_Test_Confirm : BOOL;
    CMD_Water_Valve_Test_Open : BOOL;
    CMD_Water_Valve_Test_Close : BOOL;
    CMD_Water_Valve_Test_Confirm : BOOL;
    CMD_Gas_Valve_Test_Open : BOOL;
    CMD_Gas_Valve_Test_Close : BOOL;
    CMD_Gas_Valve_Test_Confirm : BOOL;
    CMD_Water_Selective_Recover : BOOL;
    CMD_Gas_Selective_Recover : BOOL;
END_VAR

(* ---- GVL_COMMAND_POLICY_CONFIG.gvl ---- *)
{attribute 'qualified_only'}
VAR_GLOBAL
    // Command Arbitration safety policy configuration.
    // Used by PRG_Command_Arbitration only.

    // PLC inactive fail-safe policy.
    G_PLC_Inactive_Close_Gas : BOOL := TRUE;
    G_PLC_Inactive_Stop_Boiler : BOOL := TRUE;
    G_PLC_Inactive_Block_Heating : BOOL := TRUE;
    G_PLC_Inactive_Stop_Vent : BOOL := TRUE;
    G_PLC_Inactive_Block_Water : BOOL := TRUE;

    // FIRE policy.
    G_Fire_Block_Heating : BOOL := TRUE;
    G_Fire_Stop_Boiler : BOOL := TRUE;
    G_Fire_Open_Lock_1 : BOOL := TRUE;
    G_Fire_Open_Lock_2 : BOOL := TRUE;
    G_Fire_Open_Gate : BOOL := TRUE;
    G_Fire_Open_Wicket : BOOL := TRUE;
    G_Fire_Block_Lock_Close : BOOL := TRUE;

    // GAS policy.
    G_Gas_Close_Gas : BOOL := TRUE;
    G_Gas_Stop_Boiler : BOOL := TRUE;
    G_Gas_Block_Heating : BOOL := TRUE;
    G_Gas_Open_Gate : BOOL := TRUE;
    G_Gas_Open_Wicket : BOOL := TRUE;
    // Intentionally FALSE by project decision: Lock 1/2 are not evacuation contour for GAS.
    G_Gas_Open_Lock_1 : BOOL := FALSE;
    G_Gas_Open_Lock_2 : BOOL := FALSE;

    // WATER policy.
    G_Water_Block_Water : BOOL := TRUE;

    // GLOBAL_STOP policy.
    G_GlobalStop_Block_Heating : BOOL := TRUE;
    G_GlobalStop_Stop_Boiler : BOOL := TRUE;
    G_GlobalStop_Stop_Vent : BOOL := TRUE;
    G_GlobalStop_Block_Water : BOOL := TRUE;

    // Sanity policy.
    G_Block_Close_When_Open_Commanded : BOOL := TRUE;
END_VAR

(* ---- GVL_COMMAND_SHADOW.gvl ---- *)
VAR_GLOBAL
    // Operational command layer produced by PRG_Command_Arbitration during migration.
    // Used by downstream execution consumers and PRG_IO_Write.

    // Gas / boiler / ventilation
    G_Gas_Valve_Close : BOOL := FALSE;
    G_Boiler_Stop : BOOL := FALSE;
    G_Supply_100_Req : BOOL := FALSE;
    G_Supply_80_Req : BOOL := FALSE;
    G_Vent_PV3_Boost : BOOL := FALSE;
    G_Exhaust_100_Req : BOOL := FALSE;
    G_Vent_Stop : BOOL := FALSE;
    G_Vent_Block : BOOL := FALSE;
    G_Vent_Smoke_Exhaust : BOOL := FALSE;

    // Heating domain command gates
    G_Heating_Block : BOOL := FALSE;
    G_Heating_Emergency_Stop : BOOL := FALSE;
    G_Heating_Gas_Safety_Stop : BOOL := FALSE;

    // Water domain command gates
    G_Water_Block : BOOL := FALSE;
    G_Water_Emergency_Stop : BOOL := FALSE;
    G_Close_Valve_35 : BOOL := FALSE;
    G_Close_Valve_36 : BOOL := FALSE;

    // Access / evacuation locks
    G_Lock_1_Open : BOOL := FALSE;
    G_Lock_1_Close : BOOL := FALSE;
    G_Lock_2_Open : BOOL := FALSE;
    G_Lock_2_Close : BOOL := FALSE;
    G_Gate_Open : BOOL := FALSE;
    G_Wicket_Open : BOOL := FALSE;
END_VAR

(* ---- GVL_COMMAND_VERIFY.gvl ---- *)
VAR_GLOBAL
    // ======================================================
    // COMMAND VERIFIER DIAGNOSTICS STATE
    // ======================================================
    // Post-IO diagnostics published by PRG_Command_Verifier.
    // These fields are visibility/diagnostics only and must not
    // become upstream runtime or output publication authority.
    // ======================================================

    Command_Mismatch_Count : INT := 0;
    Command_Match_OK : BOOL := TRUE;
    Command_Mismatch_Active : BOOL := FALSE;

    Runtime_Sanity_OK : BOOL := TRUE;
    Runtime_Sanity_Error_Count : UDINT := 0;
    Runtime_Last_Error_Code : UDINT := 0;
    Runtime_Last_Error_Time_MS : UDINT := 0;
    Runtime_Last_Error_Text : STRING(160) := '';

    // ======================================================
    // PRE-OUTPUT SAFETY BARRIER STATE
    // ======================================================
    // Authoritative current-cycle barrier executed before PRG_IO_Write.
    // IO_Write consumes PreOutput_Block_IO as the pre-output hard-stop gate.
    // ======================================================

    PreOutput_Barrier_OK : BOOL := TRUE;
    PreOutput_Block_IO : BOOL := FALSE;
    PreOutput_Block_Count : UDINT := 0;
    PreOutput_Last_Error_Code : UDINT := 0;
    PreOutput_Last_Error_Time_MS : UDINT := 0;
    PreOutput_Last_Error_Text : STRING(160) := '';
END_VAR

(* ---- GVL_COMPLIANCE_FEDERATION_FABRIC.gvl ---- *)
VAR_GLOBAL
    // Global deterministic compliance federation authority.
    Compliance_Federation_Valid : BOOL := FALSE;
    Compliance_Federation_Granted : BOOL := FALSE;
    Compliance_Federation_Quarantine_Active : BOOL := TRUE;

    // Cross-jurisdiction governance coherence proofs.
    Regulatory_Semantics_Coherent : BOOL := FALSE;
    Certification_Boundary_Valid : BOOL := FALSE;
    Regional_Safety_Envelope_Aligned : BOOL := FALSE;
    Governance_Trust_Boundary_Stable : BOOL := FALSE;
    Policy_Compliance_Coherent : BOOL := FALSE;

    // Federated compliance synchronization.
    CrossJurisdiction_Authority_Aligned : BOOL := FALSE;
    Compliance_Runtime_Projection_Stable : BOOL := FALSE;
    External_Governance_Interpretation_Valid : BOOL := FALSE;
    Certified_Operational_Semantics_Valid : BOOL := FALSE;

    // Regulatory semantic split-brain detectors.
    CrossJurisdiction_Semantic_Drift_Detected : BOOL := FALSE;
    Certification_Boundary_Violation_Detected : BOOL := FALSE;
    Policy_Compliance_Divergence_Detected : BOOL := FALSE;
    Regional_Safety_Envelope_Mismatch_Detected : BOOL := FALSE;
    Regulatory_Trust_Corruption_Detected : BOOL := FALSE;
    Governance_Authority_Leakage_Detected : BOOL := FALSE;

    // Federation epochs.
    Compliance_Federation_Epoch : UDINT := 0;
    Compliance_Federation_Epoch_Coherent : BOOL := FALSE;

    // Temporal authority.
    Compliance_Federation_Last_Update_MS : UDINT := 0;
    Compliance_Federation_Lease_Expired : BOOL := TRUE;

    // Diagnostics.
    Compliance_Federation_Last_Error_Code : UDINT := 0;
    Compliance_Federation_Last_Error_Text : STRING(160) := '';
    Compliance_Federation_Invalidation_Count : UDINT := 0;
END_VAR

(* ---- GVL_CONFIG.gvl ---- *)
{attribute 'qualified_only'}
VAR_GLOBAL
    // Subsystem Configurations
    G_Heating_Config : ST_Heating_Config;
    G_DHW_Config : ST_DHW_Config;
    G_Security_Config : ST_Security_Global_Config;

    // HMI Configurations
    G_HMI_FloorHeating_Configs : ARRAY[1..GVL_CONSTANTS.C_MAX_HEATING_CIRCUITS] OF ST_FloorHeating_Circuit_Config;
    G_Heating_Circuit_To_Zone : ARRAY[1..GVL_CONSTANTS.C_MAX_HEATING_CIRCUITS] OF INT := [1, 2, 3, 4, 5, 6, 7, 8, 9, 10, 11, 12, 13, 14, 15, 16];
    G_Wet_Zone_Map : ARRAY[1..32] OF BOOL;
    G_HMI_Tariff_Settings : ST_Tariff_Config;
    G_HMI_Vent_Global_Config : ST_Ventilation_Global_Config;
    G_HMI_Scenario_Configs : ARRAY[1..GVL_CONSTANTS.C_MAX_SCENARIOS] OF ST_Scenario_Config;
    G_HMI_Flood_Config : ST_Flood_Global_Config;
    G_Flood_Global_Config : ST_Flood_Global_Config;
    G_HMI_User_Rules : ARRAY[1..GVL_CONSTANTS.C_MAX_RULES] OF ST_User_Rule;

    // Sensor calibration pipeline
    G_Calib_Outdoor_Temp : ST_Sensor_Calibration_Record;
    G_Calib_Supply_Temps : ARRAY[1..GVL_CONSTANTS.C_MAX_SUPPLY_TEMPS] OF ST_Sensor_Calibration_Record;
    G_Calib_Room_Temps : ARRAY[1..GVL_CONSTANTS.C_MAX_ZONES] OF ST_Sensor_Calibration_Record;
    G_Calib_Floor_Temps : ARRAY[1..GVL_CONSTANTS.C_MAX_ZONES] OF ST_Sensor_Calibration_Record;
    G_Calib_CO2 : ARRAY[1..GVL_CONSTANTS.C_MAX_ZONES] OF ST_Sensor_Calibration_Record;
    G_Calib_Humidity : ARRAY[1..GVL_CONSTANTS.C_MAX_ZONES] OF ST_Sensor_Calibration_Record;
    G_Calib_Manifold_T_Supply : ARRAY[1..GVL_CONSTANTS.C_MAX_MANIFOLDS] OF ST_Sensor_Calibration_Record;
    G_Calib_Manifold_T_Return : ARRAY[1..GVL_CONSTANTS.C_MAX_MANIFOLDS] OF ST_Sensor_Calibration_Record;
    G_Calib_Methane : ARRAY[1..GVL_CONSTANTS.C_MAX_METHANE_SENSORS] OF ST_Sensor_Calibration_Record;
    G_Calib_CO : ARRAY[1..GVL_CONSTANTS.C_MAX_CO_SENSORS] OF ST_Sensor_Calibration_Record;

    // Valve test configuration
    G_Valve_Test_Config : ARRAY[1..GVL_CONSTANTS.C_MAX_MANIFOLDS] OF ST_Valve_Test_Config;

    // HMI Commands & States
    G_HMI_Apply_Settings : BOOL;
    G_HMI_Mute_Alarm : BOOL;
    G_HMI_Ack_Alarms : BOOL;

    // Entrance lighting assist configuration.
    // Physical lux connection is optional and can be enabled later from HMI/config.
    G_Entrance_Light_Assist_Enabled : BOOL := TRUE;
    G_Entrance_Light_Assist_Use_Lux_Sensor : BOOL := FALSE;
    G_Entrance_Light_Assist_Fallback_To_Night : BOOL := TRUE;
    G_Entrance_Light_Assist_Lux_Threshold : REAL := 50.0;
    G_Entrance_Light_Assist_Duration_MS : UDINT := 300000;
    G_Entrance_Door_1_Index : INT := 1;
    G_Entrance_Door_2_Index : INT := 2;
    G_Entrance_Corridor_Light_Zone : INT := 1;
    G_Entrance_Stairs_Light_Zone : INT := 2;
    G_Entrance_Corridor_Light_Level : BYTE := 100;
    G_Entrance_Stairs_Light_Level : BYTE := 30;

    // Access Control Commands
    G_HMI_Gate_Open_Req : BOOL;
    G_HMI_Wicket_Open_Req : BOOL;
    G_HMI_Lock_1_Open_Req : BOOL;
    G_HMI_Lock_1_Close_Req : BOOL;
    G_HMI_Lock_2_Open_Req : BOOL;
    G_HMI_Lock_2_Close_Req : BOOL;
    G_Access_Pulse_MS : UDINT := 500;

    // Network security
    G_Allowed_IPs : ARRAY[1..GVL_CONSTANTS.C_MAX_ALLOWED_IPS] OF STRING(15) := ['192.168.1.100','192.168.1.101','127.0.0.1','',''];

    G_Backup_Circulation_Pump_In_Service : BOOL := TRUE;
    G_Electric_Heater_In_Service : BOOL := TRUE;
    G_Freeze_Hardware_Retry_Count : INT := 2;
    G_Freeze_Hardware_Retry_Delay_MS : UDINT := 5000;
    G_Pump_Exercise_Enabled : BOOL := TRUE;
    G_Pump_Exercise_Interval_MS : UDINT := 604800000;
    G_Pump_Exercise_Duration_MS : UDINT := 30000;
    G_Manifold_Pump_In_Service : ARRAY[1..GVL_CONSTANTS.C_MAX_MANIFOLDS] OF BOOL := [TRUE, TRUE, TRUE, TRUE, TRUE];
    G_Manifold_Priority : ARRAY[1..GVL_CONSTANTS.C_MAX_MANIFOLDS] OF INT := [3, 3, 2, 2, 1];
    G_Manifold_Thermal_Weight : ARRAY[1..GVL_CONSTANTS.C_MAX_MANIFOLDS] OF REAL := [1.0, 1.0, 0.8, 0.8, 0.5];
    G_Max_Active_Manifolds : INT := 3;
    G_Max_Thermal_Budget : REAL := 6.0;
    G_Policy_Min_Hold_MS : UDINT := 300000;
    G_DHW_Heating_Pump_In_Service : BOOL := TRUE;
    G_DHW_Circ_Pump_In_Service : BOOL := TRUE;
    G_Water_Valve_Exercise_Enabled : BOOL := TRUE;
    G_Water_Valve_Exercise_Interval_MS : UDINT := 604800000;
    G_Water_Valve_Exercise_Duration_MS : UDINT := 15000;
    G_Water_Valve_Close_Retry_Count : INT := 2;
    G_Water_Valve_Close_Retry_Delay_MS : UDINT := 3000;

    // OpenTherm / Modbus adapter configuration
    G_OpenTherm_Enabled : BOOL := FALSE;
    G_OpenTherm_Heartbeat_Timeout_MS : UDINT := 5000;
    G_OpenTherm_Command_Ack_Timeout_MS : UDINT := 3000;
    G_OpenTherm_Register_Map : ARRAY[1..GVL_CONSTANTS.C_MAX_BOILERS] OF ST_OpenTherm_Register_Map;

    // Modbus RTU transport configuration
    // Scalar fields are used instead of nested structure for CODESYS/build-system compatibility.
    G_Modbus_RTU_Driver_Attached : BOOL := FALSE;
    G_Modbus_RTU_Port_Number : BYTE := 1; // 1=COM1, 2=COM2, 3=COM3, 4=COM4
    G_Modbus_RTU_Baudrate : UDINT := 9600;
    G_Modbus_RTU_Parity : BYTE := 1; // 0=None, 1=Even, 2=Odd
    G_Modbus_RTU_Stop_Bits : BYTE := 1; // 1 or 2
    G_Modbus_RTU_Data_Bits : BYTE := 8; // usually 8
    G_Modbus_RTU_Slave_ID : BYTE := 1;
    G_Modbus_RTU_Poll_Interval_MS : UDINT := 100;
    G_Modbus_RTU_Request_Timeout_MS : UDINT := 250;
    G_Modbus_RTU_Retry_Count : INT := 2;

    // IO Mapping
    G_FloorTemp_Map : ARRAY[1..GVL_CONSTANTS.C_MAX_HEATING_CIRCUITS] OF INT := [1, 2, 3, 4, 5, 6, 7, 8, 9, 10, 11, 12, 13, 14, 15, 16];
    G_RoomTemp_Map : ARRAY[1..16] OF INT := [1, 2, 3, 4, 5, 6, 7, 8, 9, 10, 11, 12, 13, 14, 15, 16];
    G_Door_Map : ARRAY[1..GVL_CONSTANTS.C_MAX_DOOR_SENSORS] OF INT := [1, 2, 3, 4, 5, 6, 7, 8];
    G_Window_Map : ARRAY[1..16] OF INT := [9, 10, 11, 12, 13, 14, 15, 16, 17, 18, 19, 20, 21, 22, 23, 24];

    // Evacuation config
    C_MAX_LIGHT_ZONES : INT := 32;
    G_Evac_Exit_Zones : ARRAY[1..32] OF BOOL;
    G_Evac_Zone_Names : ARRAY[1..32] OF STRING(80);

END_VAR

VAR_GLOBAL CONSTANT
    C_MS_PER_SEC : UDINT := GVL_CONSTANTS.C_MS_IN_SECOND;
    C_SEC_PER_MIN : UDINT := 60;
    C_MIN_PER_HOUR : UDINT := 60;
    C_MS_PER_MIN : UDINT := GVL_CONSTANTS.C_MS_IN_MINUTE;
    C_MAX_RULES : INT := 20;
    C_ZONE_COUNT : BYTE := 18;

    ERR_PRESSURE_OUT_OF_RANGE : UDINT := 16#E004;
    ERR_HIGH_DELTA_T : UDINT := 16#E005;
    ERR_BOILER_OFFLINE : UDINT := 16#E006;
    ERR_BOILER_GENERAL_FAULT : UDINT := 16#E007;
    ERR_BOILER_NO_FLAME : UDINT := 16#E008;
    ERR_PUMP_NO_CURRENT : UDINT := 16#E009;
    ERR_PUMP_UNDERCURRENT : UDINT := 16#E00A;
    ERR_PUMP_OVERCURRENT : UDINT := 16#E00B;
    ERR_DELTA_T_LOW : UDINT := 16#E00C;
    ERR_DELTA_T_HIGH : UDINT := 16#E00D;
    ERR_DHW_IO_OFFLINE : UDINT := 16#E00E;
    ERR_DHW_TEMP_SENSOR_FAULT : UDINT := 16#E00F;
    ERR_DHW_PRESSURE_OUT_OF_RANGE : UDINT := 16#E010;
    ERR_DHW_PRESSURE_SENSOR_FAULT : UDINT := 16#E011;
    ERR_BACKUP_PUMP_OUT_OF_SERVICE : UDINT := 16#E012;
    ERR_ELECTRIC_HEATER_OUT_OF_SERVICE : UDINT := 16#E013;
    ERR_MANIFOLD_PUMP_OUT_OF_SERVICE : UDINT := 16#E014;
    ERR_DHW_HEATING_PUMP_OUT_OF_SERVICE : UDINT := 16#E015;
    ERR_DHW_CIRC_PUMP_OUT_OF_SERVICE : UDINT := 16#E016;
    ERR_FREEZE_HARDWARE_FAILED : UDINT := 16#E017;
END_VAR

(* ---- GVL_Config_Activation.gvl ---- *)
{attribute 'qualified_only'}
VAR_GLOBAL RETAIN
    G_Requested_Config_Version : UDINT;
    G_Staged_Config_Version : UDINT;
    G_Last_Stable_Config_Version : UDINT;

    G_Activation_Request : BOOL;
    G_Rollback_Request : BOOL;

    G_Staged_Topology_Config : ARRAY[1..64] OF ST_Water_Topology_Config_Record;
END_VAR

VAR_GLOBAL
    G_Activation_State : ST_Config_Activation_State;

    G_Config_Quarantine_Active : BOOL;
    G_Activation_Runtime_Valid : BOOL;
    G_Last_Update_MS : UDINT;

    G_Status_Code : UINT;
    G_Status_Text : STRING(160);
END_VAR

(* ---- GVL_CONFIG_BACKUP.gvl ---- *)
{attribute 'qualified_only'}
VAR_GLOBAL
    // Full runtime snapshot of configuration values that can be restored
    // after validation or calibration faults. File/gateway archival remains
    // a separate porting-stage concern via GVL_FILE_ARCHIVE.

    G_Backup_FloorHeating_Configs : ARRAY[1..GVL_CONSTANTS.C_MAX_HEATING_CIRCUITS] OF ST_FloorHeating_Circuit_Config;

    G_Backup_Max_Active_Manifolds : INT := 0;
    G_Backup_Max_Thermal_Budget : REAL := 0.0;

    // Sensor calibration backup. Calibration records are configuration data:
    // invalid active calibration must be recoverable by PRG_Config_Versioning.
    G_Backup_Calib_Outdoor_Temp : ST_Sensor_Calibration_Record;
    G_Backup_Calib_Ambient_Lux : ST_Sensor_Calibration_Record;
    G_Backup_Calib_Supply_Temps : ARRAY[1..GVL_CONSTANTS.C_MAX_SUPPLY_TEMPS] OF ST_Sensor_Calibration_Record;
    G_Backup_Calib_Room_Temps : ARRAY[1..GVL_CONSTANTS.C_MAX_ZONES] OF ST_Sensor_Calibration_Record;
    G_Backup_Calib_Floor_Temps : ARRAY[1..GVL_CONSTANTS.C_MAX_ZONES] OF ST_Sensor_Calibration_Record;
    G_Backup_Calib_CO2 : ARRAY[1..GVL_CONSTANTS.C_MAX_ZONES] OF ST_Sensor_Calibration_Record;
    G_Backup_Calib_Humidity : ARRAY[1..GVL_CONSTANTS.C_MAX_ZONES] OF ST_Sensor_Calibration_Record;
    G_Backup_Calib_Manifold_T_Supply : ARRAY[1..GVL_CONSTANTS.C_MAX_MANIFOLDS] OF ST_Sensor_Calibration_Record;
    G_Backup_Calib_Manifold_T_Return : ARRAY[1..GVL_CONSTANTS.C_MAX_MANIFOLDS] OF ST_Sensor_Calibration_Record;
    G_Backup_Calib_Methane : ARRAY[1..GVL_CONSTANTS.C_MAX_METHANE_SENSORS] OF ST_Sensor_Calibration_Record;
    G_Backup_Calib_CO : ARRAY[1..GVL_CONSTANTS.C_MAX_CO_SENSORS] OF ST_Sensor_Calibration_Record;

    // Integrity flag
    G_Backup_Valid : BOOL := FALSE;
END_VAR

(* ---- GVL_CONFIG_CONTROL.gvl ---- *)
{attribute 'qualified_only'}
VAR_GLOBAL
    // Config change control. HMI/service writes here, never directly to active safety config.

    G_Apply_Request : BOOL := FALSE;
    G_Apply_Confirm : BOOL := FALSE;
    G_Rollback_Request : BOOL := FALSE;
    G_Rollback_Confirm : BOOL := FALSE;
    G_Reset_Default_Request : BOOL := FALSE;
    G_Reset_Default_Confirm : BOOL := FALSE;

    G_Config_Version : UDINT := 1;
    G_Last_Good_Version : UDINT := 1;
    G_Staged_Config_Version : UDINT := 1;
    G_Staged_Last_Changed_MS : UDINT := 0;
    G_Backup_Valid : BOOL := FALSE;
    G_Apply_Done : BOOL := FALSE;
    G_Rollback_Done : BOOL := FALSE;

    // STAGED INPUT CONFIG
    STG_Reputation_Learning_Rate : REAL := 0.05;
    STG_Reputation_Recovery_Decay : REAL := 0.01;
    STG_Min_Sensor_Confidence : REAL := 0.1;
    STG_Bad_Spike_Confidence : REAL := 0.3;
    STG_Default_Confidence : REAL := 1.0;

    // STAGED SCENARIO CONFIG
    STG_Night_Start_Hour : INT := 22;
    STG_Night_End_Hour : INT := 6;
    STG_VentBoost_Humidity_Threshold : REAL := 65.0;

    // STAGED RECOVERY CONFIG
    STG_Stabilization_Delay_MS : UDINT := 5000;

    // STAGED COMMAND POLICY CRITICAL PART
    STG_PLC_Inactive_Close_Gas : BOOL := TRUE;
    STG_PLC_Inactive_Stop_Boiler : BOOL := TRUE;
    STG_PLC_Inactive_Block_Heating : BOOL := TRUE;
    STG_PLC_Inactive_Stop_Vent : BOOL := TRUE;
    STG_PLC_Inactive_Block_Water : BOOL := TRUE;

    // BACKUP INPUT CONFIG
    BCK_Reputation_Learning_Rate : REAL := 0.05;
    BCK_Reputation_Recovery_Decay : REAL := 0.01;
    BCK_Min_Sensor_Confidence : REAL := 0.1;
    BCK_Bad_Spike_Confidence : REAL := 0.3;
    BCK_Default_Confidence : REAL := 1.0;

    // BACKUP SCENARIO CONFIG
    BCK_Night_Start_Hour : INT := 22;
    BCK_Night_End_Hour : INT := 6;
    BCK_VentBoost_Humidity_Threshold : REAL := 65.0;

    // BACKUP RECOVERY CONFIG
    BCK_Stabilization_Delay_MS : UDINT := 5000;

    // BACKUP COMMAND POLICY CRITICAL PART
    BCK_PLC_Inactive_Close_Gas : BOOL := TRUE;
    BCK_PLC_Inactive_Stop_Boiler : BOOL := TRUE;
    BCK_PLC_Inactive_Block_Heating : BOOL := TRUE;
    BCK_PLC_Inactive_Stop_Vent : BOOL := TRUE;
    BCK_PLC_Inactive_Block_Water : BOOL := TRUE;
END_VAR

(* ---- GVL_CONFIG_HISTORY.gvl ---- *)
{attribute 'qualified_only'}
VAR_GLOBAL
    // History (ring buffer of last 5 versions)
    G_History_Version : ARRAY[1..5] OF UDINT;
    G_History_Time_MS : ARRAY[1..5] OF UDINT;
    G_History_Action : ARRAY[1..5] OF STRING(64);

    G_History_Index : INT := 1;

    // Audit
    G_Last_Changed_By_Level : INT := 0;
    G_Last_Action_Text : STRING(128) := '';
END_VAR

(* ---- GVL_CONFIG_SIMULATION.gvl ---- *)
{attribute 'qualified_only'}
VAR_GLOBAL
    G_Simulation_Request : BOOL := FALSE;
    G_Simulation_Confirm : BOOL := FALSE;
    G_Simulation_Result_OK : BOOL := TRUE;
    G_Simulation_Error_Text : STRING(200) := '';
    G_Simulation_Last_Run_MS : UDINT := 0;
    G_Simulation_Result_Seq : UDINT := 0;
    G_Simulation_Staged_Config_Version : UDINT := 0;
END_VAR

(* ---- GVL_CONFIG_VALIDATION.gvl ---- *)
{attribute 'qualified_only'}
VAR_GLOBAL
    G_Config_Valid : BOOL := TRUE;
    G_Config_Critical_Error : BOOL := FALSE;
    G_Config_Force_Safe_Mode : BOOL := TRUE;
    G_Config_Auto_Corrected : BOOL := FALSE;
    G_Config_Reset_To_Default_Done : BOOL := FALSE;
    G_Config_Active_Error_Text : STRING(200) := '';
    G_Config_Control_Error_Text : STRING(200) := '';
    G_Config_Last_Error_Text : STRING(200) := '';
    G_Config_Last_Action_Text : STRING(200) := '';
    G_Config_Last_Update_MS : UDINT := 0;
END_VAR

(* ---- GVL_Config_Versioning.gvl ---- *)
{attribute 'qualified_only'}
VAR_GLOBAL
    // Versioning
    G_Config_Current_Version : UDINT := 1;
    G_Config_Last_Good_Version : UDINT := 1;

    // Checksums (simple placeholder, can be replaced with CRC)
    G_Config_Current_Checksum : UDINT := 0;
    G_Config_Last_Good_Checksum : UDINT := 0;

    // Rollback flags
    G_Config_Rollback_Requested : BOOL := FALSE;
    G_Config_Rollback_Active : BOOL := FALSE;
    G_Config_Invalid_Detected : BOOL := FALSE;
END_VAR

(* ---- GVL_CONSTANTS.gvl ---- *)
{attribute 'qualified_only'}
VAR_GLOBAL CONSTANT
    // Размеры массивов (конфигурация системы)
    C_MAX_ZONES            : INT := 16;
    C_MAX_LIGHTING_ZONES   : INT := 32;
    C_MAX_HEATING_CIRCUITS : INT := 16;
    C_MAX_CLIMATE_ZONES    : INT := 16;
    C_MAX_LIGHT_ZONES      : INT := 32;
    C_MAX_SOCKETS          : INT := 36;
    C_MAX_BLINDS           : INT := 20;
    C_MAX_ALARMS           : INT := 20;
    C_MAX_RULES            : INT := 20;
    C_MAX_MANIFOLDS        : INT := 5;
    C_MAX_BOILERS          : INT := 2;
    C_MAX_SUPPLY_FANS      : INT := 3;
    C_MAX_EXHAUST_FANS     : INT := 5;
    C_MAX_SECURITY_SENSORS : INT := 15;
    C_MAX_FLOOD_SENSORS    : INT := 12;
    C_MAX_DOOR_SENSORS     : INT := 8;
    C_MAX_CO_SENSORS       : INT := 8;
    C_MAX_METHANE_SENSORS  : INT := 2;
    C_PRIMARY_METHANE_SENSOR_INDEX : INT := 1;
    C_PRIMARY_EFFECTIVE_GAS_INDEX : INT := 1;
    C_MAX_VENT_UNITS       : INT := 8;
    C_MAX_SUPPLY_TEMPS     : INT := 2;
    C_MAX_SMOKE_SENSORS    : INT := 6;
    C_MAX_SCENARIOS        : INT := 6;
    C_MAX_OUTDOOR_ZONES    : INT := 4;
    C_MAX_ACCESS_CODES     : INT := 10;
    C_MAX_WET_ZONES        : INT := 4;
    C_MAX_CALIBRATIONS     : INT := 20;
    C_MAX_MODULES          : INT := 10;
    C_MAX_CLEANING_MODES   : INT := 3;
    C_MAX_ALLOWED_IPS      : INT := 5;
    C_MAX_VENT_SUPPLY_MODES: INT := 3;
    C_MAX_SECURITY_PHONES  : INT := 5;
    // Flood isolation groups: 1-3 local risers, 4 common inlet 35/36.
    C_MAX_FLOOD_VALVES     : INT := 4;
    C_MAX_HUMIDITY_SENSORS : INT := 8;
    C_MAX_CO2_SENSORS      : INT := 8;
    C_MAX_CIRCUITS_PER_MANIFOLD : INT := 4;
    C_MAX_TREND_DATA_POINTS: INT := 100;
    C_MAX_HISTORY_RECORDS  : INT := 100;
    C_MAX_DEBUG_LOGS       : INT := 1000;
    C_MAX_GATEWAY_COMMANDS : INT := 10;
    C_MAX_STATE_SNAPSHOTS  : INT := 10;
    // Runtime blackbox depth. The buffer is RAM-only; CSV/file archive is
    // connected later during porting/module selection.
    C_MAX_BLACKBOX_RECORDS : INT := 32;
    C_MAX_PRESENCE_HISTORY : INT := 1008;
    C_MAX_MODBUS_REGISTERS : INT := 201;
    C_MAX_DEDUPLICATION_HISTORY : INT := 100;
    // Compact retained operational mirror. Legacy 100x128 NVRAM reservation is removed.
    C_NVRAM_COMPACT_BYTES  : INT := 512;

    C_MAX_WATER_ZONES      : INT := 32;

    C_ANALOG_RAW_MAX       : WORD := 27648;
    C_ANALOG_4MA_RAW       : WORD := 5529;
    C_ANALOG_3_6MA_RAW     : WORD := 4976;
    C_ANALOG_21MA_RAW      : WORD := 29030;
    C_ANALOG_10V_MAX_RAW   : WORD := 30000;

    C_MS_IN_SECOND         : UDINT := 1000;
    C_MS_IN_MINUTE         : UDINT := 60000;
    C_MS_IN_HOUR           : UDINT := 3600000;
    C_MS_IN_DAY            : UDINT := 86400000;

    C_BOILER_CASCADE_MIN_DEMAND : REAL := 25.0;
    C_BOILER_CASCADE_HIGH_DEMAND : REAL := 250.0;
    C_BOILER_SETPOINT_MIN : REAL := 35.0;
    C_BOILER_SETPOINT_MAX : REAL := 55.0;
    C_MIN_HEATING_MANIFOLD_PRESSURE : REAL := 0.8;
END_VAR

(* ---- GVL_CONVERGENCE.gvl ---- *)
VAR_GLOBAL
    Recovery_Stable_Cycle_Count : UDINT := 0;
    Recovery_Stable_Time_MS : UDINT := 0;
    Convergence_Healthy_Observed : BOOL := FALSE;
    Convergence_Lease_OK : BOOL := FALSE;
    Convergence_Release_Allowed : BOOL := FALSE;
    Convergence_Oscillation_Quarantine_Active : BOOL := FALSE;
    Convergence_Last_Healthy_MS : UDINT := 0;
    Convergence_Last_Invalidation_MS : UDINT := 0;
    Convergence_Invalidation_Count : UDINT := 0;
    Convergence_Min_Stable_Cycles : UDINT := 5;
    Convergence_Min_Stable_Time_MS : UDINT := 500;
    Convergence_Runtime_Barrier_OK : BOOL := FALSE;
    Convergence_Runtime_Snapshot_OK : BOOL := FALSE;
    Convergence_Distributed_Snapshot_OK : BOOL := FALSE;
    Convergence_Distributed_Commit_OK : BOOL := FALSE;
    Convergence_Semantic_Progress_OK : BOOL := FALSE;
    Convergence_Output_Freshness_OK : BOOL := FALSE;
    Convergence_Last_Error_Code : UDINT := 0;
    Convergence_Last_Error_Text : STRING(160) := '';
END_VAR

(* ---- GVL_DEBUG.gvl ---- *)
{attribute 'qualified_only'}
VAR_GLOBAL
    G_Device_Health_Zones : ARRAY[1..GVL_CONSTANTS.C_MAX_CLIMATE_ZONES] OF ST_Device_Health;
    G_Device_Health_Manifolds : ARRAY[1..GVL_CONSTANTS.C_MAX_MANIFOLDS] OF ST_Device_Health;
    G_Device_Health_Boilers : ARRAY[1..GVL_CONSTANTS.C_MAX_BOILERS] OF ST_Device_Health;
    G_Device_Health_Vents : ARRAY[1..GVL_CONSTANTS.C_MAX_MANIFOLDS] OF ST_Device_Health;
    G_System_Health_Summary : BYTE := 100;
    G_Pump_Health : ARRAY[1..GVL_CONSTANTS.C_MAX_MANIFOLDS] OF ST_Device_Health; // Для 5 коллекторных насосов
    G_Gas_Valve_Health : ST_Device_Health;
END_VAR
